(* IEC 61131-3 sources: plc_simulator/services/codesys/POUs (part 8) *)

(* ---- FB_STC_MainScheduler.st ---- *)
(* ===========================================================================================
 *  FB_STC_MainScheduler — Master scheduler orchestrator
 *
 *  Company : Galvatek part of the John Cockerill Group
 *  Author  : Jarmo Piipponen
 *  Created : 25.03.2026
 *
 * -------------------------------------------------------------------------------------------
 *  Manages FB_TSK_Scheduler and FB_DEP_Scheduler calls on
 *  alternating PLC scan cycles. Ensures they never execute
 *  on the same cycle.
 *
 *  Synchronization rules:
 *  1. Normal: alternate TSK_TURN → DEP_TURN → TSK_TURN
 *  2. Skip DEP when TSK is still computing (vPhase < 10000)
 *  3. Skip DEP when gDepPending.Valid = TRUE
 *  4. gTskStable is computed after each TSK call
 *
 *  Turn values: 0=INIT, 1=TSK_TURN, 2=DEP_TURN
 *
 *  ------------------------------------------------------------------------------------------
 *
 *  Changes:
 *
 *
 *
 *)

FUNCTION_BLOCK FB_STC_MainScheduler

(* Introduction of Variables ----------------------------------------------------------------*)

VAR_INPUT
  iRun   : BOOL;     (* TRUE = run *)
  iTimeS : LINT;     (* current absolute time (s), unix seconds *)
END_VAR

VAR_EXTERNAL CONSTANT
  MAX_UNITS     : INT;
  NOT_PROCESSED : INT;
END_VAR

VAR_EXTERNAL
  gTskStable              : BOOL;
  gConflictResolved       : BOOL;
  gDepPending             : UDT_JC_DepPendingWriteType;
  gBatch                  : ARRAY[1..MAX_UNITS] OF UDT_BatchType;
  gSchedule               : ARRAY[1..MAX_UNITS] OF UDT_JC_TskScheduleType;
  gDepWkSchedule          : ARRAY[1..MAX_UNITS] OF UDT_JC_TskScheduleType;
  (* Scheduler debug globals — written here, read by Gateway via OPC UA *)
  gSchedDbgTskPhase       : INT;
  gSchedDbgDepPhase       : INT;
  gSchedDbgTurn           : INT;
  gSchedDbgSkipCnt        : INT;
  gSchedDbgDepRejectCnt   : INT;
  gSchedDbgDepFitRound    : INT;
  gSchedDbgDepCurWaitUnit : INT;
  gSchedDbgDepWaitCnt     : INT;
  gSchedDbgBatchCnt       : INT;
  gSchedDbgTskRoundTicks  : INT;
  gSchedDbgDepRoundTicks  : INT;
END_VAR

VAR_OUTPUT
  oTskPhase : INT;     (* TSK scheduler vPhase *)
  oDepPhase : INT;     (* DEP scheduler vPhase *)
  oTurn     : INT;     (* 1=TSK ran, 2=DEP ran *)
  oSkipCnt  : INT;     (* DEP skipped count (debug) *)
END_VAR

VAR
  vFB_TskScheduler  : FB_TSK_Scheduler;
  vFB_DepScheduler  : FB_DEP_Scheduler;
  vFB_TwaCalcLimits : FB_TWA_CalcLimits;
  (* dispatch — now FC FC_STC_DispatchTask, no instance vNeeded *)
  vTurn             : INT := 0;   (* 0=init, 1=TSK, 2=DEP *)
  vSkipCnt          : INT := 0;
  vTskPhase         : INT := 0;
  vUi               : INT;
END_VAR

IF NOT iRun THEN
  (* Stop both schedulers *)
  vFB_TskScheduler(iRun := FALSE, iTimeS := 0);
  vFB_DepScheduler(iRun := FALSE, iTimeS := 0, iTskPhase := 0);
  vTurn := 0;
  vTskPhase := 0;
  oTskPhase := 0;
  oDepPhase := 0;
  oTurn := 0;
  RETURN;
END_IF;

(* ── Calculate transporter working areas (X-limits) every cycle ── *)
vFB_TwaCalcLimits();

(* ── Dispatch tasks to idle transporters (every scan) ── *)
FC_STC_DispatchTask();

(* ── Determine this cycle's vTurn ── *)
IF vTurn = 0 THEN
  (* First scan: always start with TSK *)
  vTurn := 1;

ELSIF vTurn = 1 THEN
  (* Last cycle was TSK → normally DEP's vTurn *)
  (* But skip DEP if: *)
  (*   a) TSK has not reached READY yet (vPhase < 10000) *)
  (*   b) pending data waiting for TSK to process *)
  IF vTskPhase < 10000 THEN
    (* TSK still computing — DEP would be blocked at WAIT_STABLE *)
    vTurn := 1;
    vSkipCnt := vSkipCnt + 1;
  ELSIF gDepPending.Valid THEN
    (* TSK must process pending before DEP continues *)
    vTurn := 1;
    vSkipCnt := vSkipCnt + 1;
  ELSE
    vTurn := 2;
  END_IF;

ELSIF vTurn = 2 THEN
  (* Last cycle was DEP → TSK's vTurn.
     DEP now works on sandbox arrays g_dep_wk_xxx, never live globals,
     so TSK can run freely on any cycle. *)
  vTurn := 1;
END_IF;

(* ── Execute the selected scheduler ── *)
IF vTurn = 1 THEN
  (* TSK vTurn *)
  vFB_TskScheduler(iRun := TRUE, iTimeS := iTimeS);
  vTskPhase := vFB_TskScheduler.oPhase;

  (* JS parity: set stable only when TSK reached READY and conflictResolved; do not clear here *)
    IF (vTskPhase >= 10000) AND gConflictResolved THEN
      gTskStable := TRUE;
  END_IF;

ELSIF vTurn = 2 THEN
  (* DEP vTurn *)
  vFB_DepScheduler(
    iRun       := TRUE,
    iTimeS    := iTimeS,
    iTskPhase := vTskPhase
  );
END_IF;

(* ── Publish waiting batch schedules from DEP workspace for UI display ── *)
FOR vUi := 1 TO MAX_UNITS DO
  IF gBatch[vUi].State = NOT_PROCESSED AND gDepWkSchedule[vUi].StageCount > 0 THEN
    gSchedule[vUi] := gDepWkSchedule[vUi];
  END_IF;
END_FOR;

(* ── Update outputs ── *)
oTskPhase := vFB_TskScheduler.oPhase;
oDepPhase := vFB_DepScheduler.oPhase;
oTurn      := vTurn;
oSkipCnt  := vSkipCnt;

(* ── Forward to scheduler debug globals (OPC UA readable) ── *)
gSchedDbgTskPhase        := vFB_TskScheduler.oPhase;
gSchedDbgDepPhase        := vFB_DepScheduler.oPhase;
gSchedDbgTurn             := vTurn;
gSchedDbgSkipCnt         := vSkipCnt;
gSchedDbgDepRejectCnt   := vFB_DepScheduler.oRejectCnt;
gSchedDbgDepFitRound    := vFB_DepScheduler.oFitRound;
gSchedDbgDepCurWaitUnit := vFB_DepScheduler.oCurWaitUnit;
gSchedDbgDepWaitCnt     := vFB_DepScheduler.oWaitCnt;
gSchedDbgBatchCnt        := vFB_TskScheduler.oBatchCnt;
gSchedDbgTskRoundTicks  := vFB_TskScheduler.oRoundTicks;
gSchedDbgDepRoundTicks  := vFB_DepScheduler.oRoundTicks;

END_FUNCTION_BLOCK

(* ---- FB_TSK_Scheduler.st ---- *)
(* ===========================================================================================
 *  FB_TSK_Scheduler — Main task scheduler state machine
 *
 *  Company : Galvatek part of the John Cockerill Group
 *  Author  : Jarmo Piipponen
 *  Created : 25.03.2026
 *
 * -------------------------------------------------------------------------------------------
 *  One vPhase per PLC scan cycle.
 *
 *  Phase flow (structured by 100/1000 groups):
 *  0        STOPPED
 *  1        INIT             (collect active batches)
 *  2        NO_TREATMENT_STATES
 *  1000+i   CALC_SCHEDULE    (schedule for batch i, 0..vBatchCount-1)
 *  2000     CLEAR_TASKS      (clear task queues)
 *  2001+i   CREATE_TASKS     (tasks for batch i, 0..vBatchCount-1)
 *  2100     SORT_TASKS
 *  2101     SWAP_TASKS
 *  2102     ANALYZE          (→ 2103 if vConflict, → 2200 if clean)
 *  2103     RESOLVE          (→ 2100 loop, or → 2200 if max iter)
 *  2200     NO_TREATMENT     (create no-treatment tasks)
 *  2201     APPLY_STRETCHES  (persist resolve decisions)
 *  10000    READY            (cycle complete)
 *  10001    CHECK_DEP_PENDING
 *  10002    RESTART          (→ 1)
 *
 *  Phase advancement:
 *  Default = vPhase + 1 (at end of function body).
 *  vNextPhase is set ONLY when jumping to a different group.
 *
 *  Conflict resolution: one vConflict per cycle.
 *  If resolved → back to SORT (2100).
 *  If no vConflict → NO_TREATMENT → READY.
 *  Max iterations to prevent infinite loops.
 *
 *  ------------------------------------------------------------------------------------------
 *
 *  Changes:
 *  25.03.2026 - Restructured: vPhase+1 default, vIdx from vPhase offset.
 *
 *
 *)

FUNCTION_BLOCK FB_TSK_Scheduler

(* Introduction of Variables ----------------------------------------------------------------*)

VAR_INPUT
  iRun                     : BOOL;    (* TRUE = run, FALSE = stop *)
  iTimeS                  : LINT;    (* current absolute time (s), unix seconds *)
END_VAR

VAR_EXTERNAL CONSTANT
    MAX_TRANSPORTERS        : INT;
    MAX_UNITS               : INT;
    MAX_LOCKS               : INT;
END_VAR

VAR_EXTERNAL
  g_batch                   : ARRAY[1..MAX_UNITS] OF UDT_BatchType;
  g_unit                    : ARRAY[1..MAX_UNITS] OF UDT_JC_UnitType;
  TreatmentPrograms                 : ARRAY[1..MAX_UNITS] OF UDT_TreatmentProgramType;
  g_task                    : ARRAY[1..MAX_TRANSPORTERS] OF UDT_JC_TskQueueType;
  g_schedule                : ARRAY[1..MAX_UNITS] OF UDT_JC_TskScheduleType;
  Transporters                     : ARRAY[0..MAX_TRANSPORTERS] OF UDT_TransporterType;
  (* DEP handshake *)
  g_dep_pending             : UDT_JC_DepPendingWriteType;
  g_conflict_resolved       : BOOL;
  g_tsk_stable              : BOOL;
  (* Debug observability *)
  g_dbg_tsk_conflict_type   : INT;
  g_dbg_tsk_conflict_iter   : INT;
  g_dbg_tsk_conf_unit       : INT;
  g_dbg_tsk_conf_stage      : INT;
  g_dbg_tsk_blocked_unit    : INT;
  g_dbg_tsk_blocked_stage   : INT;
  g_dbg_tsk_deficit         : DINT;
  g_dbg_tsk_stretch_cnt     : INT;
  g_dbg_tsk_total_adv       : DINT;
  g_dbg_tsk_total_delay     : DINT;
  g_dbg_prog_cal            : ARRAY[1..MAX_UNITS] OF DINT;
END_VAR

VAR_OUTPUT
  oPhase                   : INT;
  oBatchCnt               : INT;
  oTaskCnt                : INT;
  oCycleCnt               : INT;
  oConflict                : BOOL;
  oRoundTicks             : INT;     (* ticks consumed by last completed vRound *)
END_VAR

VAR
  vPhase                     : INT := 0;
  vNextPhase                : INT;
  vIdx                       : INT;    (* derived from vPhase offset *)
  (* Batch list *)
  vBatchList                : ARRAY[1..MAX_UNITS] OF INT;
  vBatchCount               : INT;
  (* Conflict iteration *)
  vConflictIter             : INT;
  MAX_CONFLICT_ITER         : INT := 40;
  (* Analyze result cache *)
  an_conflict               : BOOL;
  an_conf_type              : INT;
  an_conf_unit              : INT;
  an_conf_stage             : INT;
  an_conf_trans             : INT;
  an_blocked_unit           : INT;
  an_blocked_stage          : INT;
  an_deficit                : REAL;
  (* Resolve result cache *)
  rs_total_adv              : REAL;
  rs_total_delay            : REAL;
  (* Transporter assignment *)
  vSchedTrans               : INT;
  (* Locked stages — prevents oscillation in resolve loop *)
  vLocks                     : ARRAY[1..MAX_LOCKS] OF UDT_JC_TskLockType;
  vLockCnt                  : INT := 0;
  vLocksInitialized         : BOOL := FALSE;
  vFB_FindTransporter                   : FB_STC_FindTransporter;
  (* candidateStretches — JS: resolve decisions persisted to TreatmentPrograms *)
  vStretches                 : ARRAY[1..20] OF UDT_JC_TskStretchType;
  vStretchCnt               : INT := 0;
  si                        : INT;
  vNewCal                   : DINT;
  vFlexCap                  : DINT;
  (* Temp *)
  ui                        : INT;
  ui2                       : INT;
  ti                        : INT;
  bi                        : INT;
  vTotalTasks               : INT;
  cycle_count               : INT := 0;
  round_ticks               : INT := 0;  (* ticks since last RESTART *)
END_VAR

IF NOT iRun THEN
  IF vPhase <> 0 THEN
    FOR ti := 1 TO MAX_TRANSPORTERS DO
      g_task[ti].Count := 0;
    END_FOR;
  END_IF;
  vPhase := 0;
  oPhase := 0;
  RETURN;
END_IF;

vNextPhase := 0;
round_ticks := round_ticks + 1;

(* ══════════════════════════════════════════════════════════════ *)
(* PHASE 0: STOPPED                                             *)
(* ══════════════════════════════════════════════════════════════ *)
IF vPhase = 0 THEN
  vNextPhase := 1;

(* ══════════════════════════════════════════════════════════════ *)
(* PHASE 1: INIT — collect active batches                       *)
(* ══════════════════════════════════════════════════════════════ *)
ELSIF vPhase = 1 THEN
  (* Clear schedule for ALL units — start from clean slate *)
  FOR ui := 1 TO MAX_UNITS DO
    g_schedule[ui].StageCount := 0;
  END_FOR;
  vBatchCount := FC_STC_CollectActiveBatches(iMode := 0, oList => vBatchList);
  oBatchCnt := vBatchCount;
  vConflictIter := 0;
  vLocksInitialized := FALSE;
  vStretchCnt := 0;
  g_dbg_tsk_total_adv   := 0;
  g_dbg_tsk_total_delay := 0;

  IF vBatchCount = 0 THEN
    FOR ti := 1 TO MAX_TRANSPORTERS DO
      g_task[ti].Count := 0;
    END_FOR;
    g_conflict_resolved := TRUE;
    vNextPhase := 2200;   (* skip to NO_TREATMENT *)
  ELSE
    g_conflict_resolved := FALSE;
    (* vPhase + 1 → 2 *)
  END_IF;

(* ══════════════════════════════════════════════════════════════ *)
(* PHASE 2: NO_TREATMENT_STATES                                *)
(* ══════════════════════════════════════════════════════════════ *)
ELSIF vPhase = 2 THEN
  FC_STC_NoTreatmentStates();
  vNextPhase := 1000;

(* ══════════════════════════════════════════════════════════════ *)
(* PHASE 1000+i: CALC_SCHEDULE — one batch per scan             *)
(*   i = 0..vBatchCount-1: calculate schedule                   *)
(*   i >= vBatchCount: vDone → 2000                              *)
(* ══════════════════════════════════════════════════════════════ *)
ELSIF vPhase >= 1000 AND vPhase <= 1999 THEN
  vIdx := vPhase - 1000;

  IF vIdx < vBatchCount THEN
    ui := vBatchList[vIdx + 1];

    (* CalcSchedule handles elapsed-time normalisation — no pre-adjustment vNeeded here. *)

    IF g_unit[ui].vLocation < MIN_STATION_INDEX THEN
      vSchedTrans := g_unit[ui].vLocation;
    ELSE
      vFB_FindTransporter(iLiftStn := g_unit[ui].vLocation, iSinkStn := 0);
      vSchedTrans := vFB_FindTransporter.oTrans;
      IF vSchedTrans = 0 THEN vSchedTrans := 1; END_IF;
    END_IF;

    FC_STC_CalcSchedule(iUnit := ui, iTrans := vSchedTrans, iTimeS := iTimeS,
                     ioSchedule := g_schedule, ioBatch := g_batch, ioProgram := TreatmentPrograms);
    (* vPhase + 1 → next batch *)

  ELSE
    vNextPhase := 2000;
  END_IF;

(* ══════════════════════════════════════════════════════════════ *)
(* PHASE 2000: CLEAR_TASKS — clear all task queues              *)
(* ══════════════════════════════════════════════════════════════ *)
ELSIF vPhase = 2000 THEN
  FOR ti := 1 TO MAX_TRANSPORTERS DO
    g_task[ti].Count := 0;
  END_FOR;
  (* vPhase + 1 → 2001 *)

(* ══════════════════════════════════════════════════════════════ *)
(* PHASE 2001+i: CREATE_TASKS — one batch per scan              *)
(*   i = 0..vBatchCount-1: create tasks                         *)
(*   i >= vBatchCount: vDone → 2100                              *)
(* ══════════════════════════════════════════════════════════════ *)
ELSIF vPhase >= 2001 AND vPhase <= 2099 THEN
  vIdx := vPhase - 2001;

  IF vIdx < vBatchCount THEN
    ui := vBatchList[vIdx + 1];
    FC_STC_CreateTasks(iUnit := ui, ioSchedule := g_schedule, ioTask := g_task);
    (* vPhase + 1 → next batch *)
  ELSE
    vNextPhase := 2100;
  END_IF;

(* ══════════════════════════════════════════════════════════════ *)
(* PHASE 2100: SORT_TASKS                                       *)
(* ══════════════════════════════════════════════════════════════ *)
ELSIF vPhase = 2100 THEN
  FC_STC_SortTasks(iTrans := 0, iTimeS := iTimeS, ioTask := g_task, ioBatch := g_batch);
  IF NOT vLocksInitialized THEN
    vLockCnt := 0;
    FOR bi := 1 TO MAX_LOCKS DO
      vLocks[bi].Unit := 0;
      vLocks[bi].Stage := 0;
      vLocks[bi].Direction := 0;
    END_FOR;
    vLocksInitialized := TRUE;
  END_IF;
  (* vPhase + 1 → 2101 *)

(* ══════════════════════════════════════════════════════════════ *)
(* PHASE 2101: SWAP_TASKS                                       *)
(* ══════════════════════════════════════════════════════════════ *)
ELSIF vPhase = 2101 THEN
  FC_STC_SwapTasks(ioTask := g_task);
  (* vPhase + 1 → 2102 *)

(* ══════════════════════════════════════════════════════════════ *)
(* PHASE 2102: ANALYZE                                          *)
(* ══════════════════════════════════════════════════════════════ *)
ELSIF vPhase = 2102 THEN
  FC_TSK_Analyze(ioTask := g_task,
    oHasConflict => an_conflict, oConfType => an_conf_type,
    oConfUnit => an_conf_unit, oConfStage => an_conf_stage,
    oConfTrans => an_conf_trans, oBlockedUnit => an_blocked_unit,
    oBlockedStage => an_blocked_stage, oDeficit => an_deficit);
  oConflict := an_conflict;

  IF an_conflict THEN
    g_dbg_tsk_conflict_type  := an_conf_type;
    g_dbg_tsk_conf_unit      := an_conf_unit;
    g_dbg_tsk_conf_stage     := an_conf_stage;
    g_dbg_tsk_blocked_unit   := an_blocked_unit;
    g_dbg_tsk_blocked_stage  := an_blocked_stage;
    g_dbg_tsk_deficit        := REAL_TO_DINT(an_deficit);
    g_conflict_resolved := FALSE;
    (* vPhase + 1 → 2103 RESOLVE *)
  ELSE
    g_conflict_resolved := TRUE;
    vNextPhase := 2200;   (* skip RESOLVE → NO_TREATMENT *)
  END_IF;

(* ══════════════════════════════════════════════════════════════ *)
(* PHASE 2103: RESOLVE — one vConflict, then re-analyze          *)
(* ══════════════════════════════════════════════════════════════ *)
ELSIF vPhase = 2103 THEN
  FC_TSK_Resolve(
    iConfUnit     := an_conf_unit,
    iConfStage    := an_conf_stage,
    iConfTrans    := an_conf_trans,
    iBlockedUnit  := an_blocked_unit,
    iBlockedStage := an_blocked_stage,
    iDeficit       := an_deficit,
    ioLocks        := vLocks,
    ioLockCnt     := vLockCnt,
    ioSchedule     := g_schedule,
    ioTask         := g_task,
    ioBatch        := g_batch,
    oTotalAdv     => rs_total_adv,
    oTotalDelay   => rs_total_delay
  );

  (* Collect vStretches *)
  IF rs_total_adv > 0.1 AND vStretchCnt < 20 THEN
    vStretchCnt := vStretchCnt + 1;
    vStretches[vStretchCnt].Unit   := an_blocked_unit;
    vStretches[vStretchCnt].Stage  := an_blocked_stage;
    vStretches[vStretchCnt].DelayS := -REAL_TO_DINT(rs_total_adv);
    g_dbg_tsk_total_adv := g_dbg_tsk_total_adv + REAL_TO_DINT(rs_total_adv);
  END_IF;
  IF rs_total_delay > 0.1 AND vStretchCnt < 20 THEN
    vStretchCnt := vStretchCnt + 1;
    vStretches[vStretchCnt].Unit   := an_conf_unit;
    vStretches[vStretchCnt].Stage  := an_conf_stage;
    vStretches[vStretchCnt].DelayS := REAL_TO_DINT(rs_total_delay);
    g_dbg_tsk_total_delay := g_dbg_tsk_total_delay + REAL_TO_DINT(rs_total_delay);
  END_IF;

  vConflictIter := vConflictIter + 1;

  IF vConflictIter >= MAX_CONFLICT_ITER THEN
    g_conflict_resolved := TRUE;
    vNextPhase := 2200;   (* accept partial, move on *)
  ELSE
    vNextPhase := 2100;   (* re-SORT → SWAP → ANALYZE *)
  END_IF;

(* ══════════════════════════════════════════════════════════════ *)
(* PHASE 2200: NO_TREATMENT — create no-treatment tasks         *)
(* ══════════════════════════════════════════════════════════════ *)
ELSIF vPhase = 2200 THEN
  FC_STC_ManualTask(iTimeS := iTimeS, ioTask := g_task);
  FC_TSK_NoTreatment(iTimeS := iTimeS, ioTask := g_task);
  oConflict := FALSE;
  (* vPhase + 1 → 2201 *)

(* ══════════════════════════════════════════════════════════════ *)
(* PHASE 2201: APPLY_STRETCHES — persist resolve decisions      *)
(* ══════════════════════════════════════════════════════════════ *)
ELSIF vPhase = 2201 THEN
  FOR si := 1 TO vStretchCnt DO
    IF vStretches[si].Unit >= 1 AND vStretches[si].Unit <= MAX_UNITS THEN
     IF vStretches[si].Stage >= 1
        AND vStretches[si].Stage <= TreatmentPrograms[vStretches[si].Unit].StepCount THEN
      vNewCal := TreatmentPrograms[vStretches[si].Unit].Steps[vStretches[si].Stage].CalTime
               + vStretches[si].DelayS;
      IF vNewCal < TreatmentPrograms[vStretches[si].Unit].Steps[vStretches[si].Stage].MinTime THEN
        vNewCal := TreatmentPrograms[vStretches[si].Unit].Steps[vStretches[si].Stage].MinTime;
      END_IF;
      (* Flex cap: min + factor × (max - min) *)
      vFlexCap := TreatmentPrograms[vStretches[si].Unit].Steps[vStretches[si].Stage].MinTime
               + REAL_TO_DINT(SCH_TSK_FLEX_FACTOR * DINT_TO_REAL(
                   TreatmentPrograms[vStretches[si].Unit].Steps[vStretches[si].Stage].MaxTime
                 - TreatmentPrograms[vStretches[si].Unit].Steps[vStretches[si].Stage].MinTime));
      IF vNewCal > vFlexCap THEN
        vNewCal := vFlexCap;
      END_IF;
      TreatmentPrograms[vStretches[si].Unit].Steps[vStretches[si].Stage].CalTime := vNewCal;

      IF g_batch[vStretches[si].Unit].CurStage = vStretches[si].Stage THEN
        g_batch[vStretches[si].Unit].CalTime := vNewCal;
      END_IF;
     END_IF;
    END_IF;
  END_FOR;
  vStretchCnt := 0;
  (* vPhase + 1 → 2202 *)

(* ══════════════════════════════════════════════════════════════ *)
(* PHASE 2202: MOVE_AWAY — idle transporter move-away check     *)
(* ══════════════════════════════════════════════════════════════ *)
ELSIF vPhase = 2202 THEN
  FC_STC_TakeOut(iTimeS := iTimeS);
  vNextPhase := 10000;

(* ══════════════════════════════════════════════════════════════ *)
(* PHASE 10000: READY — cycle complete                          *)
(* ══════════════════════════════════════════════════════════════ *)
ELSIF vPhase = 10000 THEN
  vTotalTasks := 0;
  FOR ti := 1 TO MAX_TRANSPORTERS DO
    vTotalTasks := vTotalTasks + g_task[ti].Count;
  END_FOR;
  oTaskCnt := vTotalTasks;

  IF NOT oConflict THEN
    g_dbg_tsk_conflict_type := 0;
    g_dbg_tsk_conf_unit     := 0;
    g_dbg_tsk_conf_stage    := 0;
    g_dbg_tsk_blocked_unit  := 0;
    g_dbg_tsk_blocked_stage := 0;
    g_dbg_tsk_deficit       := 0;
  END_IF;
  g_dbg_tsk_conflict_iter := vConflictIter;
  g_dbg_tsk_stretch_cnt   := vStretchCnt;

  FOR ui := 1 TO MAX_UNITS DO
    IF g_batch[ui].CurStage >= 1
       AND g_batch[ui].CurStage <= TreatmentPrograms[ui].StepCount THEN
      g_dbg_prog_cal[ui] := TreatmentPrograms[ui].Steps[g_batch[ui].CurStage].CalTime;
    ELSE
      g_dbg_prog_cal[ui] := 0;
    END_IF;
  END_FOR;
  (* vPhase + 1 → 10001 *)

(* ══════════════════════════════════════════════════════════════ *)
(* PHASE 10001: CHECK_DEP_PENDING                               *)
(* ══════════════════════════════════════════════════════════════ *)
ELSIF vPhase = 10001 THEN
  IF g_dep_pending.Valid THEN
    FOR ui := 1 TO MAX_UNITS DO
      IF g_dep_pending.Programs[ui].ProgramId > 0 THEN
        TreatmentPrograms[ui] := g_dep_pending.Programs[ui];
      END_IF;
    END_FOR;
    IF g_dep_pending.BatchUnit >= 1 AND g_dep_pending.BatchUnit <= MAX_UNITS THEN
      g_batch[g_dep_pending.BatchUnit].CurStage   := g_dep_pending.BatchStage;
      g_batch[g_dep_pending.BatchUnit].State       := g_dep_pending.BatchState;
      g_batch[g_dep_pending.BatchUnit].StartTime   := g_dep_pending.TimeStamp;
      g_batch[g_dep_pending.BatchUnit].MinTime     := g_dep_pending.BatchMinTime;
      g_batch[g_dep_pending.BatchUnit].MaxTime     := g_dep_pending.BatchMaxTime;
      g_batch[g_dep_pending.BatchUnit].CalTime     := g_dep_pending.BatchCalTime;
    END_IF;
    (* Apply active batch CalTimes written by DEP *)
    FOR ui := 1 TO MAX_UNITS DO
      IF g_dep_pending.ActiveBatchCalTime[ui] > 0
         AND ui <> g_dep_pending.BatchUnit THEN
        g_batch[ui].CalTime := g_dep_pending.ActiveBatchCalTime[ui];
      END_IF;
    END_FOR;
    g_dep_pending.Valid := FALSE;
    g_conflict_resolved := FALSE;
    g_tsk_stable := FALSE;
    vNextPhase := 1;   (* full recalculation *)
  END_IF;
  (* else vPhase + 1 → 10002 *)

(* ══════════════════════════════════════════════════════════════ *)
(* PHASE 10002: RESTART — begin new cycle                       *)
(* ══════════════════════════════════════════════════════════════ *)
ELSIF vPhase = 10002 THEN
  cycle_count := cycle_count + 1;
  oCycleCnt := cycle_count;
  oRoundTicks := round_ticks;
  round_ticks := 0;
  vNextPhase := 1;

(* ══════════════════════════════════════════════════════════════ *)
(* Unknown vPhase → reset                                        *)
(* ══════════════════════════════════════════════════════════════ *)
ELSE
  vNextPhase := 1;
END_IF;

(* ── Phase advancement: default = vPhase + 1 ── *)
IF vNextPhase > 0 THEN
  vPhase := vNextPhase;
ELSE
  vPhase := vPhase + 1;
END_IF;
oPhase := vPhase;

END_FUNCTION_BLOCK

(* ---- FB_TWA_CalcLimits.st ---- *)
(* ===========================================================================================
 *  FB_TWA_CalcLimits — Transporter Working Area: X-limit calculation
 *
 *  Company : Galvatek part of the John Cockerill Group
 *  Author  : Jarmo Piipponen
 *  Created : 25.03.2026
 *
 * -------------------------------------------------------------------------------------------
 *  Calculates x_min_limit and x_max_limit for all active
 *  transporters. Collision avoidance layers:
 *
 *  Pass 1 (per transporter):
 *  - Station restrictions from gAvoidStatus
 *  - Safety vDistance from same-line neighbors
 *  - canEvade, vPriority, x-vRank computation
 *
 *  Pass 2 (pair comparisons):
 *  - Priority-based restrictions (higher → lower)
 *  - Bidirectional safety (same direction chase)
 *
 *  Final: Trap validation
 *
 *  ------------------------------------------------------------------------------------------
 *
 *  Changes:
 *
 *
 *
 *)

FUNCTION_BLOCK FB_TWA_CalcLimits

(* Introduction of Variables ----------------------------------------------------------------*)

VAR_EXTERNAL CONSTANT
    MAX_TRANSPORTERS  : INT;
    MAX_UNITS         : INT;
    MIN_STATION_INDEX : INT;
    MAX_STATION_INDEX : INT;
    AVOID_PASSABLE    : INT;
    AVOID_BLOCK       : INT;
    MIN_WORKING_AREA  : DINT;
    IN_PROCESS        : INT;
END_VAR

VAR_EXTERNAL
  Transporters      : ARRAY[0..MAX_TRANSPORTERS] OF UDT_TransporterType;
  gTransporter      : ARRAY[1..MAX_TRANSPORTERS] OF UDT_TransporterStatusType;
  Stations          : ARRAY[MIN_STATION_INDEX..MAX_STATION_INDEX] OF UDT_StationType;
  CountStations     : INT;
  gAvoidStatus      : ARRAY[MIN_STATION_INDEX..MAX_STATION_INDEX] OF INT;
  gStationOccupancy : ARRAY[1..MAX_STATION_INDEX] OF UDT_JC_UnitAtStationType;
  gBatch            : ARRAY[1..MAX_UNITS] OF UDT_BatchType;
END_VAR

VAR
  i             : INT;
  j             : INT;
  vStnNum       : INT;
  vStnX         : DINT;
  vAvoidSt      : INT;
  vMinX         : DINT;
  vMaxX         : DINT;
  vCurrentX     : DINT;
  vCurrentY     : DINT;
  vAvoidDist    : DINT;
  vIsTarget     : BOOL;
  vNewVal       : DINT;

  (* Station scan: nearest restricting station per side *)
  vNearLeftX    : DINT;
  vNearLeftStn  : INT;
  vNearRightX   : DINT;
  vNearRightStn : INT;
  vHasLeft      : BOOL;
  vHasRight     : BOOL;
  vMidpoint     : DINT;

  (* Per-transporter computed values *)
  vPriority     : ARRAY[1..MAX_TRANSPORTERS] OF DINT;
  vCanEvade     : ARRAY[1..MAX_TRANSPORTERS] OF BOOL;
  vRank         : ARRAY[1..MAX_TRANSPORTERS] OF INT;

  (* Pair comparison *)
  vOtherX       : DINT;
  vOtherY       : DINT;
  vIPhase       : INT;
  vJPhase       : INT;
  vDist         : DINT;
  vWorkArea     : DINT;
  vAWins        : BOOL;
  vRestrictX    : DINT;
  vBetween      : INT;
  vChainOfs     : DINT;
  vAdjusted     : DINT;

  (* Bidirectional *)
  vIMovingRight : BOOL;
  vIMovingLeft  : BOOL;
  vJMovingRight : BOOL;
  vJMovingLeft  : BOOL;

  (* IN_PROCESS batch vPriority boost *)
  vLiftStn      : INT;
  vLiftUid      : INT;
  vBatchBoost   : DINT;

  (* Full task extent for vRestrictX *)
  vLiftX        : DINT;
  vSinkX        : DINT;
  vILiftStn     : INT;
  vISinkStn     : INT;
END_VAR

(* ══════════════════════════════════════════════════════════════
   PASS 1: Station restrictions + safety vDistance + properties
   Each transporter computes its OWN limits in one iteration.
   ══════════════════════════════════════════════════════════════ *)
FOR i := 1 TO MAX_TRANSPORTERS DO
  IF NOT gTransporter[i].IsActive THEN
    vPriority[i] := 0;
    vCanEvade[i] := FALSE;
    vRank[i] := 0;
    CONTINUE;
  END_IF;

  vMinX := Transporters[i].DrivePosMin;
  vMaxX := Transporters[i].DrivePosMax;
  vCurrentX := gTransporter[i].XPosition;
  vCurrentY := gTransporter[i].YPosition;
  vAvoidDist := Transporters[i].AvoidanceWidth;

  (* Lock transporters with no drive range configured *)
  IF (vMinX < 1) OR (vMaxX < 1) THEN
    gTransporter[i].XMinDriveLimit := vCurrentX;
    gTransporter[i].XMaxDriveLimit := vCurrentX;
    vPriority[i] := 0;
    vCanEvade[i] := FALSE;
    vRank[i] := 0;
    CONTINUE;
  END_IF;

  (* ── Station scan: find nearest restrict LEFT and RIGHT ──────
     Single pass through all stations. Only Block and
     Passable-target stations cause restrictions. *)
  vHasLeft := FALSE;
  vHasRight := FALSE;
  vNearLeftX := 0;
  vNearLeftStn := 0;
  vNearRightX := 0;
  vNearRightStn := 0;

  FOR vStnNum := MIN_STATION_INDEX TO MAX_STATION_INDEX DO
    IF Stations[vStnNum].TankId = 0 THEN CONTINUE; END_IF;

    vAvoidSt := gAvoidStatus[vStnNum];
    IF vAvoidSt = 0 THEN CONTINUE; END_IF;  (* AVOID_NONE *)

    (* Passable: only restricts if this transporter's target *)
    IF vAvoidSt = AVOID_PASSABLE THEN
      vIsTarget := (vStnNum = gTransporter[i].LiftStationTarget)
               OR  (vStnNum = gTransporter[i].SinkStationTarget);
      IF NOT vIsTarget THEN CONTINUE; END_IF;
    END_IF;

    (* Station is Block or Passable+target → track nearest per side *)
    vStnX := Stations[vStnNum].XPosition;

    IF vStnX < vCurrentX THEN
      IF NOT vHasLeft OR vStnX > vNearLeftX THEN
        vNearLeftX := vStnX;
        vNearLeftStn := vStnNum;
        vHasLeft := TRUE;
      END_IF;
    ELSIF vStnX > vCurrentX THEN
      IF NOT vHasRight OR vStnX < vNearRightX THEN
        vNearRightX := vStnX;
        vNearRightStn := vStnNum;
        vHasRight := TRUE;
      END_IF;
    END_IF;
  END_FOR;

  (* Apply station restrictions using station-specific AvoidDistance *)
  IF vHasLeft THEN
    vNewVal := vNearLeftX + Stations[vNearLeftStn].AvoidDistance;
    IF vNewVal > vMinX THEN vMinX := vNewVal; END_IF;
  END_IF;
  IF vHasRight THEN
    vNewVal := vNearRightX - Stations[vNearRightStn].AvoidDistance;
    IF vNewVal < vMaxX THEN vMaxX := vNewVal; END_IF;
  END_IF;

  (* Conflict: trapped vBetween two restricting stations *)
  IF (vMinX >= vMaxX) AND vHasLeft AND vHasRight THEN
    vMidpoint := (vNearLeftX + vNearRightX) / 2;
    vMinX := vMidpoint - 5;
    vMaxX := vMidpoint + 5;
  END_IF;

  (* ── Safety vDistance: each same-line neighbor pushes i away ── *)
  FOR j := 1 TO MAX_TRANSPORTERS DO
    IF j = i THEN CONTINUE; END_IF;
    IF NOT gTransporter[j].IsActive THEN CONTINUE; END_IF;

    vOtherY := gTransporter[j].YPosition;
    IF ABS(vOtherY - vCurrentY) >= 1 THEN CONTINUE; END_IF;

    vOtherX := gTransporter[j].XPosition;

    IF vOtherX < vCurrentX THEN
      (* j is LEFT → j's safety zone pushes i's min up *)
      vNewVal := vOtherX + Transporters[j].AvoidanceWidth;
  IF vNewVal > vMinX THEN vMinX := vNewVal; END_IF;
    ELSIF vOtherX > vCurrentX THEN
      (* j is RIGHT → j's safety zone pushes i's max down *)
      vNewVal := vOtherX - Transporters[j].AvoidanceWidth;
  IF vNewVal < vMaxX THEN vMaxX := vNewVal; END_IF;
    END_IF;
  END_FOR;

  (* ── Write limits ── *)
  gTransporter[i].XMinDriveLimit := vMinX;
  gTransporter[i].XMaxDriveLimit := vMaxX;

  (* ── canEvade (inline) ── *)
  vCanEvade[i] := TRUE;
  IF gTransporter[i].Status < 3 THEN
    vCanEvade[i] := FALSE;
  END_IF;
  IF (gTransporter[i].Status = 4)
     AND ((gTransporter[i].Phase = 2) OR (gTransporter[i].Phase = 4)) THEN
    vCanEvade[i] := FALSE;
  END_IF;
  vWorkArea := vMaxX - vMinX;
  IF vWorkArea < MIN_WORKING_AREA THEN
    vCanEvade[i] := FALSE;
  END_IF;

  (* ── Priority (inline, replaces TWA_CalcPriority call) ──────
     IN_PROCESS batch boost: +100000 if the task serves an
     IN_PROCESS batch. Phases 1-4 all check via LiftStation
     unit lookup (unit stays associated throughout transfer).
     This ensures treatment tasks trump NTT/empty moves. ── *)
  vIPhase := gTransporter[i].Phase;
  vBatchBoost := 0;
  IF vIPhase >= 1 AND vIPhase <= 4 THEN
    vLiftStn := gTransporter[i].LiftStationTarget;
    IF vLiftStn >= 1 AND vLiftStn <= MAX_STATION_INDEX THEN
      vLiftUid := gStationOccupancy[vLiftStn].UnitId;
      IF vLiftUid >= 1 AND vLiftUid <= MAX_UNITS THEN
        IF gBatch[vLiftUid].State = IN_PROCESS THEN
          vBatchBoost := DINT#100000;
        END_IF;
      END_IF;
    END_IF;
  END_IF;

  IF NOT vCanEvade[i] THEN
    vPriority[i] := DINT#100000;
  ELSIF vIPhase = 3 OR vIPhase = 4 THEN
    vDist := ABS(vCurrentX - gTransporter[i].XFinalTarget);
  IF vDist > 99999 THEN vDist := 99999; END_IF;
    vPriority[i] := DINT#200000 + vBatchBoost + (DINT#99999 - vDist);
  ELSIF vIPhase = 1 OR vIPhase = 2 THEN
    (* Move-away (Status=3, Phase=1) gets idle-class vPriority, not active-task vPriority *)
    IF gTransporter[i].Status = 3 THEN
      vPriority[i] := 2;  (* above stationary idle (1), below active tasks (100000+) *)
    ELSE
      vDist := ABS(vCurrentX - gTransporter[i].XFinalTarget);
      IF vDist > 99999 THEN vDist := 99999; END_IF;
      vPriority[i] := DINT#100000 + vBatchBoost + (DINT#99999 - vDist);
    END_IF;
  ELSE
    vPriority[i] := 1;
  END_IF;

  (* ── X-vRank among same-line active transporters ──
     vRank = 1 + count of same-line transporters with smaller x *)
  vRank[i] := 1;
  FOR j := 1 TO MAX_TRANSPORTERS DO
    IF j = i THEN CONTINUE; END_IF;
    IF NOT gTransporter[j].IsActive THEN CONTINUE; END_IF;
    IF ABS(gTransporter[j].YPosition - vCurrentY) >= 1 THEN CONTINUE; END_IF;
    IF gTransporter[j].XPosition < vCurrentX THEN
      vRank[i] := vRank[i] + 1;
    END_IF;
  END_FOR;
END_FOR;

(* ══════════════════════════════════════════════════════════════
   PASS 2: Priority restrictions + bidirectional safety
   Each pair (i,j): i restricts j if i has higher vPriority.
   ══════════════════════════════════════════════════════════════ *)
FOR i := 1 TO MAX_TRANSPORTERS DO
  IF NOT gTransporter[i].IsActive THEN CONTINUE; END_IF;
  IF vPriority[i] = 0 THEN CONTINUE; END_IF;

  vCurrentX := gTransporter[i].XPosition;
  vCurrentY := gTransporter[i].YPosition;
  vIPhase := gTransporter[i].Phase;

  FOR j := 1 TO MAX_TRANSPORTERS DO
    IF j = i THEN CONTINUE; END_IF;
    IF NOT gTransporter[j].IsActive THEN CONTINUE; END_IF;
    IF vPriority[j] = 0 THEN CONTINUE; END_IF;

    vOtherY := gTransporter[j].YPosition;
    IF ABS(vOtherY - vCurrentY) >= 1 THEN CONTINUE; END_IF;

    vOtherX := gTransporter[j].XPosition;
    vJPhase := gTransporter[j].Phase;

    (* ── Priority restrictions: i restricts j if i wins ── *)
    (* Move-away (Status=3, Phase=1) participates in restrictions
       so it can push stationary idle transporters out of its way *)
    IF (vIPhase <> 0) OR (gTransporter[i].Status = 3 AND vIPhase = 1) THEN
      vAWins := FALSE;
      IF vPriority[i] > vPriority[j] THEN
        vAWins := TRUE;
      ELSIF (vPriority[i] = vPriority[j]) AND (i < j) THEN
        vAWins := TRUE;
      END_IF;

      IF vAWins THEN
        (* Full task extent: use the extreme position
           of both lift and sink stations on the side
           facing j. This prevents j from first driving
           closer and then having to reverse when i
           moves to the other end of its task. *)
        vILiftStn := gTransporter[i].LiftStationTarget;
        vISinkStn := gTransporter[i].SinkStationTarget;
        IF vIPhase >= 1 AND vIPhase <= 4 THEN
          vLiftX := vCurrentX;
          vSinkX := vCurrentX;
          IF vILiftStn >= MIN_STATION_INDEX
             AND vILiftStn <= MAX_STATION_INDEX THEN
            vLiftX := Stations[vILiftStn].XPosition;
          END_IF;
          IF vISinkStn >= MIN_STATION_INDEX
             AND vISinkStn <= MAX_STATION_INDEX THEN
            vSinkX := Stations[vISinkStn].XPosition;
          END_IF;
          IF vCurrentX < vOtherX THEN
            (* i LEFT of j → use rightmost extent *)
            vRestrictX := vLiftX;
            IF vSinkX > vRestrictX THEN
              vRestrictX := vSinkX;
            END_IF;
            IF vCurrentX > vRestrictX THEN
              vRestrictX := vCurrentX;
            END_IF;
          ELSE
            (* i RIGHT of j → use leftmost extent *)
            vRestrictX := vLiftX;
            IF vSinkX < vRestrictX THEN
              vRestrictX := vSinkX;
            END_IF;
            IF vCurrentX < vRestrictX THEN
              vRestrictX := vCurrentX;
            END_IF;
          END_IF;
        ELSE
          vRestrictX := vCurrentX;
        END_IF;

        (* "vBetween" from pre-computed vRank *)
        vBetween := ABS(vRank[i] - vRank[j]) - 1;
  IF vBetween < 0 THEN vBetween := 0; END_IF;

        vChainOfs := Transporters[i].AvoidanceWidth
                   + INT_TO_DINT(vBetween) * (MIN_WORKING_AREA + Transporters[i].AvoidanceWidth);

        IF vCurrentX < vOtherX THEN
          (* i LEFT, j RIGHT → restrict j's XMin *)
          vNewVal := vRestrictX + vChainOfs;
          IF vNewVal > gTransporter[j].XMinDriveLimit THEN
            IF vNewVal <= (gTransporter[j].XMaxDriveLimit - MIN_WORKING_AREA) THEN
              gTransporter[j].XMinDriveLimit := vNewVal;
            ELSE
              vAdjusted := gTransporter[j].XMaxDriveLimit - MIN_WORKING_AREA;
              IF vAdjusted > gTransporter[j].XMinDriveLimit THEN
                gTransporter[j].XMinDriveLimit := vAdjusted;
              END_IF;
            END_IF;
          END_IF;

        ELSIF vCurrentX > vOtherX THEN
          (* i RIGHT, j LEFT → restrict j's XMax *)
          vNewVal := vRestrictX - vChainOfs;
          IF vNewVal < gTransporter[j].XMaxDriveLimit THEN
            IF vNewVal >= (gTransporter[j].XMinDriveLimit + MIN_WORKING_AREA) THEN
              gTransporter[j].XMaxDriveLimit := vNewVal;
            ELSE
              vAdjusted := gTransporter[j].XMinDriveLimit + MIN_WORKING_AREA;
              IF vAdjusted < gTransporter[j].XMaxDriveLimit THEN
                gTransporter[j].XMaxDriveLimit := vAdjusted;
              END_IF;
            END_IF;
          END_IF;
        END_IF;
      END_IF;
    END_IF;

    (* ── Bidirectional safety: only adjacent (vRank diff = 1) ── *)
    IF ABS(vRank[i] - vRank[j]) = 1 THEN
      vIMovingRight := ((vIPhase = 1) OR (vIPhase = 3))
                        AND (gTransporter[i].XFinalTarget > vCurrentX);
      vJMovingRight := ((vJPhase = 1) OR (vJPhase = 3))
                        AND (gTransporter[j].XFinalTarget > vOtherX);
      vIMovingLeft := ((vIPhase = 1) OR (vIPhase = 3))
                       AND (gTransporter[i].XFinalTarget < vCurrentX);
      vJMovingLeft := ((vJPhase = 1) OR (vJPhase = 3))
                       AND (gTransporter[j].XFinalTarget < vOtherX);

      IF vCurrentX < vOtherX AND vIMovingRight AND vJMovingRight THEN
        (* i LEFT chasing j RIGHT → restrict j's XMin *)
        vNewVal := vCurrentX + Transporters[i].AvoidanceWidth;
        IF vNewVal > gTransporter[j].XMinDriveLimit THEN
          gTransporter[j].XMinDriveLimit := vNewVal;
        END_IF;
      END_IF;

      IF vCurrentX > vOtherX AND vIMovingLeft AND vJMovingLeft THEN
        (* i RIGHT chasing j LEFT → restrict j's XMax *)
        vNewVal := vCurrentX - Transporters[i].AvoidanceWidth;
        IF vNewVal < gTransporter[j].XMaxDriveLimit THEN
          gTransporter[j].XMaxDriveLimit := vNewVal;
        END_IF;
      END_IF;
    END_IF;
  END_FOR;
END_FOR;

(* ══════════════════════════════════════════════════════════════
   TRAP VALIDATION: if restrictions vConflict, lock in place
   ══════════════════════════════════════════════════════════════ *)
FOR i := 1 TO MAX_TRANSPORTERS DO
  IF NOT gTransporter[i].IsActive THEN CONTINUE; END_IF;
  IF gTransporter[i].XMinDriveLimit > gTransporter[i].XMaxDriveLimit THEN
    gTransporter[i].XMinDriveLimit := gTransporter[i].XPosition;
    gTransporter[i].XMaxDriveLimit := gTransporter[i].XPosition;
  END_IF;
END_FOR;

END_FUNCTION_BLOCK

(* ---- SIM_FB_ClearConfig.st ---- *)
(* ============================================================
   SIM_FB_ClearConfig.st — Clear all PLC configuration data

   Called by PLC_PRG when Gateway sends cmd=3 (clear_all).
   Zeroes out all stations, transporter configs, transporter
   states and units so the PLC is ready for fresh config upload.
   ============================================================ *)

FUNCTION_BLOCK SIM_FB_ClearConfig
VAR_EXTERNAL CONSTANT
    MAX_Transporters    : INT;
    MAX_STATIONS_PER_STEP       : INT;
    MIN_StationIndex : INT;
    MAX_StationIndex   : INT;
    MAX_Units           : INT;
    DEP_MAX_WAITING     : INT;
END_VAR

VAR_EXTERNAL
  g_station_count    : INT;
  g_station         : ARRAY[MIN_StationIndex..MAX_StationIndex] OF UDT_StationType;
  g_station_loc     : ARRAY[1..MAX_StationIndex] OF UDT_UnitLocation;
  g_cfg              : ARRAY[1..MAX_Transporters] OF UDT_TransporterType;
  g_transporter      : ARRAY[1..MAX_Transporters] OF UDT_TransporterStatusType;
  g_sim_trans        : ARRAY[1..MAX_Transporters] OF UDT_JC_SimTransporterType;
  g_unit            : ARRAY[1..MAX_Units] OF UDT_UnitType;
  g_ntt             : ARRAY[1..MAX_Transporters] OF UDT_JC_NttTransporterType;
  g_batch          : ARRAY[1..MAX_Units] OF UDT_BatchType;
  g_program         : ARRAY[1..MAX_Units] OF UDT_TreatmentProgramType;
  g_avoid_status     : ARRAY[MIN_StationIndex..MAX_StationIndex] OF INT;
  g_schedule         : ARRAY[1..MAX_Units] OF UDT_JC_TskScheduleType;
  g_task             : ARRAY[1..MAX_Transporters] OF UDT_JC_TskQueueType;
  g_dep_sandbox      : UDT_JC_DepSandboxType;
  g_dep_pending      : UDT_JC_DepPendingWriteType;
  g_dep_activated    : BOOL;
  g_tsk_stable       : BOOL;
  g_dep_waiting_count : INT;
  g_dep_waiting       : ARRAY[1..DEP_MAX_WAITING] OF INT;
  g_dep_wait_unit     : INT;
END_VAR
VAR
  i : INT;
  j : INT;
  k : INT;
END_VAR

(* --- Clear all stations --- *)
FOR i := MIN_StationIndex TO MAX_StationIndex DO
  g_station[i].TankId       := 0;
  g_station[i].IsInUse       := FALSE;
  g_station[i].XPosition    := 0;
  g_station[i].YPosition    := 0;
  g_station[i].ZPosition    := 0;
  g_station[i].DryWet          := 0;
  g_station[i].StationType     := 0;
  g_station[i].DrippingTime := 0;
  g_station[i].DeviceDelay  := 0;
END_FOR;

(* --- Clear all location tracking (transporters 1..MAX_Transporters + stations MIN..MAX) --- *)
FOR i := 1 TO MAX_StationIndex DO
  g_station_loc[i].UnitId     := 0;
  g_station_loc[i].ChangeTime := 0;
END_FOR;
g_station_count := 0;

(* --- Clear all transporter configs --- *)
FOR i := 1 TO MAX_Transporters DO
  g_cfg[i].DrivePosMin   := 0;
  g_cfg[i].DrivePosMax   := 0;
  g_cfg[i].YMinDriveLimit   := 0;
  g_cfg[i].YMaxDriveLimit   := 0;
  g_cfg[i].CollisionWidth    := 0;
  g_cfg[i].AvoidanceWidth    := 0;
  g_cfg[i].Acceleration_X     := 0;
  g_cfg[i].Deceleration_X     := 0;
  g_cfg[i].SpeedMax_X    := 0;
  g_cfg[i].ZPosDown    := 0;
  g_cfg[i].ZPosSlowUp := 0;
  g_cfg[i].ZPosSlowDown := 0;
  g_cfg[i].ZPosSlowEnd := 0;
  g_cfg[i].SpeedLiftSlow_Z   := 0;
  g_cfg[i].SpeedLiftFast_Z   := 0;
  g_cfg[i].DripTrayDelay  := 0;
  FOR j := 1 TO 4 DO
    g_cfg[i].TaskArea[j].MinLift := 0;
    g_cfg[i].TaskArea[j].MaxLift := 0;
    g_cfg[i].TaskArea[j].MinSink := 0;
    g_cfg[i].TaskArea[j].MaxSink := 0;
  END_FOR;
END_FOR;

(* --- Clear avoid status --- *)
FOR i := MIN_StationIndex TO MAX_StationIndex DO
  g_avoid_status[i] := 0;
END_FOR;

(* --- Clear all transporter states --- *)
FOR i := 1 TO MAX_Transporters DO
  g_transporter[i].IsActive          := FALSE;
  g_transporter[i].Status          := 0;
  g_transporter[i].Phase           := 0;
  g_transporter[i].TaskId         := 0;
  g_sim_trans[i].RunningTaskId := 0;
  g_transporter[i].LiftStationTarget    := 0;
  g_transporter[i].SinkStationTarget    := 0;
  g_sim_trans[i].TreatmentTime  := 0;
  g_sim_trans[i].LiftDeviceDelay := 0;
  g_sim_trans[i].SinkDeviceDelay := 0;
  g_transporter[i].DrippingTime   := 0;
  g_transporter[i].TaskRemainingTime  := 0;
  g_transporter[i].CurrentStation := 0;
  g_transporter[i].XFinalTarget  := 0;
  g_transporter[i].XDriveTarget  := 0;
  g_transporter[i].YFinalTarget  := 0;
  g_transporter[i].YDriveTarget  := 0;
  g_transporter[i].XPosition            := 0;
  g_transporter[i].YPosition            := 0;
  g_transporter[i].ZPosition            := 0;
  g_sim_trans[i].XVelocity           := 0;
  g_sim_trans[i].ZStage         := 0;
  g_sim_trans[i].ZTimer       := 0.0;
  g_transporter[i].XMinDriveLimit     := 0;
  g_transporter[i].XMaxDriveLimit     := 0;
END_FOR;

(* --- Clear all units --- *)
FOR i := 1 TO MAX_Units DO
  g_unit[i].location := 0;
  g_unit[i].Status   := 0;
  g_unit[i].Target   := 0;
END_FOR;

(* --- Clear NTT destinations --- *)
FOR i := 1 TO MAX_Transporters DO
  FOR j := 1 TO 8 DO
    g_ntt[i].Target[j].StationCount := 0;
    g_ntt[i].Target[j].FallbackCount := 0;
    FOR k := 1 TO MAX_STATIONS_PER_STEP DO
      g_ntt[i].Target[j].Stations[k] := 0;
      g_ntt[i].Target[j].FallbackStations[k] := 0;
    END_FOR;
  END_FOR;
END_FOR;

(* --- Clear all batches --- *)
FOR i := 1 TO MAX_Units DO
  g_batch[i].BatchCode  := 0;
  g_batch[i].State       := 0;
  g_batch[i].ProgId     := 0;
  g_batch[i].CurStage   := 0;
  g_batch[i].MinTime    := 0;
  g_batch[i].MaxTime    := 0;
  g_batch[i].CalTime    := 0;
  g_batch[i].StartTime  := LINT#0;
END_FOR;

(* --- Clear all treatment programs --- *)
FOR i := 1 TO MAX_Units DO
  g_program[i].ProgramId := 0;
  g_program[i].ProgramName := '';
  g_program[i].StepCount := 0;
  FOR j := 0 TO 30 DO
    FOR k := 0 TO 4 DO
      g_program[i].Steps[j].Stations[k] := 0;
    END_FOR;
    g_program[i].Steps[j].StationCount := 0;
    g_program[i].Steps[j].MinTime := 0;
    g_program[i].Steps[j].MaxTime := 0;
    g_program[i].Steps[j].CalTime := 0;
  END_FOR;
END_FOR;

(* --- Clear all schedules (g_schedule) --- *)
FOR i := 1 TO MAX_Units DO
  g_schedule[i].StageCount := 0;
  FOR j := 1 TO 30 DO
    g_schedule[i].Stages[j].station       := 0;
    g_schedule[i].Stages[j].EntryTime    := 0;
    g_schedule[i].Stages[j].ExitTime     := 0;
    g_schedule[i].Stages[j].MinTime      := 0;
    g_schedule[i].Stages[j].CalcTime     := 0;
    g_schedule[i].Stages[j].MaxTime      := 0;
    g_schedule[i].Stages[j].TransferTime := 0;
  END_FOR;
END_FOR;

(* --- Clear all task queues (g_task) --- *)
FOR i := 1 TO MAX_Transporters DO
  g_task[i].Count := 0;
  FOR j := 1 TO 60 DO
    g_task[i].Queue[j].Unit         := 0;
    g_task[i].Queue[j].Stage        := 0;
    g_task[i].Queue[j].LiftStationTarget := 0;
    g_task[i].Queue[j].SinkStationTarget := 0;
    g_task[i].Queue[j].StartTime   := 0;
    g_task[i].Queue[j].FinishTime  := 0;
    g_task[i].Queue[j].CalcTime    := 0;
    g_task[i].Queue[j].MinTime     := 0;
    g_task[i].Queue[j].MaxTime     := 0;
  END_FOR;
END_FOR;

(* --- Clear departure sandbox and pending write --- *)
g_dep_sandbox.Valid := FALSE;
g_dep_pending.Valid := FALSE;
g_dep_pending.BatchUnit  := 0;
g_dep_pending.BatchStage := 0;
g_dep_pending.BatchState := 0;

(* --- Clear departure scheduler state (previously missing) --- *)
g_dep_activated     := FALSE;
g_tsk_stable        := TRUE;   (* JS: tasksStableFlag starts true on empty line *)
g_dep_waiting_count := 0;
g_dep_wait_unit     := 0;
FOR i := 1 TO 5 DO
  g_dep_waiting[i] := 0;
END_FOR;

END_FUNCTION_BLOCK

(* ---- SIM_FB_EventQueue.st ---- *)
(* ============================================================
   SIM_FB_EventQueue — Event message queue handler (OPC UA)
   ============================================================
   Manages a circular 10-slot event queue (g_event).

   - enqueue: caller writes msg fields to g_event_pending,
     then sets g_event_pending_valid := TRUE.
     This FB picks it up and adds to queue.
   - dequeue: Gateway reads g_event.Buffer[Head] directly
     via OPC UA, then writes g_event_ack_seq to acknowledge.
     PLC sees ack match → advance head, count--.

   Called every PLC scan from plc_prg (always, not gated by
   scheduler turn).

   OPC UA handshake:
     PLC:    g_event.Count, g_event.Head, g_event.Buffer[] → readable via OPC UA
     Gateway: g_event_ack_seq → writable via OPC UA
     When g_event_ack_seq = g_event.Buffer[Head].Seq: message consumed → next.
   ============================================================ *)

FUNCTION_BLOCK SIM_FB_EventQueue
VAR_EXTERNAL
  g_event               : UDT_JC_EventQueueType;
  g_event_pending       : UDT_JC_EventMsgType;
  g_event_pending_valid : BOOL;
  g_event_ack_seq       : INT;
END_VAR
VAR
  tail : INT;
END_VAR

(* ── 1. Enqueue: pick up pending message if queue not full ── *)
IF g_event_pending_valid AND g_event.Count < 10 THEN
  tail := ((g_event.Head - 1 + g_event.Count) MOD 10) + 1;

  g_event_pending.Seq := g_event.NextSeq;
  g_event.NextSeq := g_event.NextSeq + 1;
  IF g_event.NextSeq > 32000 THEN
    g_event.NextSeq := 1;
  END_IF;

  g_event.Buffer[tail] := g_event_pending;
  g_event.Count := g_event.Count + 1;

  g_event_pending_valid := FALSE;
END_IF;

(* ── 2. Dequeue: check gateway ack for head message ── *)
IF g_event.Count > 0 THEN
  IF g_event_ack_seq = g_event.Buffer[g_event.Head].Seq THEN
    g_event.Head := (g_event.Head MOD 10) + 1;
    g_event.Count := g_event.Count - 1;
  END_IF;
END_IF;

END_FUNCTION_BLOCK

(* ---- SIM_FB_RunTasks.st ---- *)
(* ============================================================
   SIM_FB_RunTasks.st — Simulate transporter task execution

   For each active transporter [1..3], checks whether a new task
   has been assigned (task_id <> running_task_id) and executes
   the full transport cycle:

     Phase 0  idle        — waiting for new task
     Phase 1  to_lift     — X-drive towards lift station
     Phase 2  lifting     — Z-lift sequence (stages 1-5)
     Phase 3  to_sink     — X-drive towards sink station
     Phase 4  sinking     — Z-sink sequence (stages 6-8)

   Also maintains current_station (nearest station) every cycle.

   Called once per PLC scan from PLC_PRG.
   ============================================================ *)

FUNCTION_BLOCK SIM_FB_RunTasks
VAR_INPUT
  i_run : BOOL;       (* enable — typically init_done *)
END_VAR
VAR_EXTERNAL CONSTANT
    MAX_Transporters    : INT;
    MAX_Units           : INT;
    MAX_STEPS_PER_PROGRAM          : INT;
    MIN_StationIndex : INT;
    MAX_StationIndex   : INT;
    IN_PROCESS          : INT;
END_VAR

VAR_EXTERNAL
  g_transporter  : ARRAY[1..MAX_Transporters] OF UDT_TransporterStatusType;
  g_sim_trans    : ARRAY[1..MAX_Transporters] OF UDT_JC_SimTransporterType;
  g_station     : ARRAY[MIN_StationIndex..MAX_StationIndex] OF UDT_StationType;    g_station_loc  : ARRAY[1..MAX_StationIndex] OF UDT_UnitLocation;  g_cfg          : ARRAY[1..MAX_Transporters] OF UDT_TransporterType;
  g_move         : ARRAY[1..MAX_Transporters] OF UDT_JC_MoveTimesType;
  g_actual_move  : ARRAY[1..MAX_Transporters] OF UDT_JC_ActualMoveTimeType;
  g_unit         : ARRAY[1..MAX_Units] OF UDT_UnitType;
  g_batch        : ARRAY[1..MAX_Units] OF UDT_BatchType;
  g_program      : ARRAY[1..MAX_Units] OF UDT_TreatmentProgramType;
  g_time_s       : LINT;
  g_event_pending       : UDT_JC_EventMsgType;
  g_event_pending_valid : BOOL;
END_VAR
VAR
  i            : INT;
  idx          : INT;
  (* Physics FB instances — one per transporter (MATIEC needs separate instances) *)
  fb_x1        : SIM_FB_XMotion;
  fb_x2        : SIM_FB_XMotion;
  fb_x3        : SIM_FB_XMotion;
  fb_z1        : SIM_FB_ZMotion;
  fb_z2        : SIM_FB_ZMotion;
  fb_z3        : SIM_FB_ZMotion;
  (* Station lookup — now FC STC_FindStation, no instance needed *)
  (* Temp vars for VAR_IN_OUT passing *)
  tmp_x        : DINT;
  tmp_vx       : DINT;
  tmp_z        : DINT;
  tmp_zs       : INT;
  tmp_zt       : REAL;
  arrived_x    : BOOL;
  at_station   : BOOL;    (* TRUE only when actually at station, not just at drive limit *)
  arrived_z    : BOOL;
  station_kind : INT;
  device_delay : REAL;
  drop_time    : REAL;
  pick_unit_id : INT;     (* unit_id picked up from lift station *)
  xfer_total   : REAL;    (* transfer time for UI progress bar *)
  sink_unit_id : INT;     (* unit_id being placed at sink station *)
  (* Nearest-station calculation *)
  nearest_num  : INT;
  min_dist     : DINT;
  dx           : DINT;
  (* Actual move time tracker — now FC STC_TrackMoveTimes, no instance needed *)
  (* Unit location update — now FC STC_UpdateUnitLocation, no instance needed *)
  (* Event helpers *)
  evt_unit     : INT;
  evt_diff     : LINT;
  (* Treatment time wait *)
  can_lift       : BOOL;
  lift_uid       : INT;      (* unit at lift station *)
  treat_cal      : DINT;      (* treatment cal_time for current stage *)
  treat_elapsed  : LINT;     (* seconds spent at lift station *)
  (* ── TASK_COMPLETE event: phase timestamps per transporter ── *)
  ts_task_start  : ARRAY[1..3] OF LINT;  (* Phase 0→1: task accepted *)
  ts_at_lift     : ARRAY[1..3] OF LINT;  (* Phase 1 at_station: arrived at lift *)
  ts_lift_begin  : ARRAY[1..3] OF LINT;  (* Phase 1→2: can_lift, begin lift *)
  ts_lift_done   : ARRAY[1..3] OF LINT;  (* Phase 2→3: lift complete *)
  ts_at_sink     : ARRAY[1..3] OF LINT;  (* Phase 3→4: arrived at sink *)
  (* TASK_COMPLETE temp vars *)
  dd_lift_s      : INT;   (* lift device_delay in seconds *)
  dropping_s     : INT;   (* dropping/valutus time in seconds *)
  trip_s         : INT;   (* drip tray delay in seconds, 0 if not used *)
  dur_nosto      : INT;   (* computed nosto duration *)
  dur_lasku      : INT;   (* computed lasku duration *)
END_VAR

IF NOT i_run THEN
  RETURN;
END_IF;

FOR i := 1 TO MAX_Transporters DO
  IF g_transporter[i].IsActive THEN

  (* ── Phase 0 → 1: Accept new task ───────────────────────── *)
  IF (g_transporter[i].Phase = 0)
     AND (g_transporter[i].TaskId <> g_sim_trans[i].RunningTaskId) THEN
    g_sim_trans[i].RunningTaskId := g_transporter[i].TaskId;
    g_transporter[i].XFinalTarget := STC_FindStation(station_number := g_transporter[i].LiftStationTarget);
    g_transporter[i].Phase := 1;
    STC_TrackMoveTimes(i_trans := i, i_prev := 0, i_new := 1);
    g_transporter[i].Status := 4;  (* auto_run *)
    g_sim_trans[i].ZStage := 0;
    g_sim_trans[i].ZTimer := 0.0;
    (* Record task start timestamp *)
    ts_task_start[i] := g_time_s;
    ts_at_lift[i]    := LINT#0;

  (* ── Phase 1: Drive X towards lift station ──────────────── *)
  ELSIF g_transporter[i].Phase = 1 THEN
    tmp_x  := g_transporter[i].XPosition;
    tmp_vx := g_sim_trans[i].XVelocity;
    IF i = 1 THEN
      fb_x1(
        delta_t  := 0.02,
        x_target := g_transporter[i].XFinalTarget,
        x_min    := g_transporter[i].XMinDriveLimit,
        x_max    := g_transporter[i].XMaxDriveLimit,
        v_max    := g_cfg[i].SpeedMax_X,
        t_acc    := g_cfg[i].Acceleration_X,
        t_dec    := g_cfg[i].Deceleration_X,
        x_pos    := tmp_x,
        v_x      := tmp_vx
      );
      arrived_x := fb_x1.arrived;
    ELSIF i = 2 THEN
      fb_x2(
        delta_t  := 0.02,
        x_target := g_transporter[i].XFinalTarget,
        x_min    := g_transporter[i].XMinDriveLimit,
        x_max    := g_transporter[i].XMaxDriveLimit,
        v_max    := g_cfg[i].SpeedMax_X,
        t_acc    := g_cfg[i].Acceleration_X,
        t_dec    := g_cfg[i].Deceleration_X,
        x_pos    := tmp_x,
        v_x      := tmp_vx
      );
      arrived_x := fb_x2.arrived;
    ELSIF i = 3 THEN
      fb_x3(
        delta_t  := 0.02,
        x_target := g_transporter[i].XFinalTarget,
        x_min    := g_transporter[i].XMinDriveLimit,
        x_max    := g_transporter[i].XMaxDriveLimit,
        v_max    := g_cfg[i].SpeedMax_X,
        t_acc    := g_cfg[i].Acceleration_X,
        t_dec    := g_cfg[i].Deceleration_X,
        x_pos    := tmp_x,
        v_x      := tmp_vx
      );
      arrived_x := fb_x3.arrived;
    END_IF;
    g_transporter[i].XPosition  := tmp_x;
    g_sim_trans[i].XVelocity := tmp_vx;

    (* Only transition when actually at station, not just at drive limit *)
    at_station := arrived_x
                  AND (ABS(g_transporter[i].XPosition - g_transporter[i].XFinalTarget) <= 6);
    IF at_station THEN
      g_transporter[i].CurrentStation := g_transporter[i].LiftStationTarget;
      (* Record arrival at lift station (first time only) *)
      IF ts_at_lift[i] = LINT#0 THEN
        ts_at_lift[i] := g_time_s;
      END_IF;

      (* ── Wait for treatment time AND device_delay before lifting ──
         Z-movement starts when the LONGER of two has elapsed:
         1. Remaining treatment time (unit must finish treatment)
         2. Station device_delay (covers must be open)
         Both timers run simultaneously from transporter arrival.
         This matches JS behavior: max(treatment, device_delay). *)
      can_lift := TRUE;
      STC_FindStation(station_number := g_transporter[i].LiftStationTarget, device_delay_s => device_delay, dropping_time_s => drop_time);

      (* Check treatment time *)
      lift_uid := g_station_loc[g_transporter[i].LiftStationTarget].UnitId;
      IF lift_uid >= 1 AND lift_uid <= MAX_Units THEN
        IF g_batch[lift_uid].State = IN_PROCESS
           AND g_batch[lift_uid].CurStage >= 1
           AND g_batch[lift_uid].CurStage <= MAX_STEPS_PER_PROGRAM THEN
          treat_cal := g_program[lift_uid].Steps[g_batch[lift_uid].CurStage].CalTime;
          IF treat_cal > 0 THEN
            treat_elapsed := g_time_s - g_station_loc[g_transporter[i].LiftStationTarget].ChangeTime;
            IF treat_elapsed < DINT_TO_LINT(treat_cal) THEN
              can_lift := FALSE;
            END_IF;
          END_IF;
        END_IF;
      END_IF;

      (* Check device_delay — covers must have had time to open since arrival *)
      IF can_lift AND device_delay > 0.0 THEN
        IF LINT_TO_REAL(g_time_s - ts_at_lift[i]) < device_delay THEN
          can_lift := FALSE;
        END_IF;
      END_IF;

      IF can_lift THEN
      (* Record lift begin timestamp *)
      ts_lift_begin[i] := g_time_s;
      (* drop_time already captured by STC_FindStation above *)
      (* Skip stage 1 — device_delay already overlapped above.
         Z-movement starts immediately (stage 2).
         dropping_time and drip_tray_delay happen at the TOP. *)
      g_transporter[i].ZPosition := 0;
      g_sim_trans[i].ZTimer := 0.0;
      g_sim_trans[i].ZStage := 2;
      g_transporter[i].Phase := 2;
      STC_TrackMoveTimes(i_trans := i, i_prev := 1, i_new := 2);

      (* ── Calculate transfer time (used by event + batch times) ── *)
      xfer_total := STC_CalcTransferTime(
        i_from_stn            := g_transporter[i].LiftStationTarget,
        i_to_stn              := g_transporter[i].SinkStationTarget,
        i_move                := g_move[i],
        i_from_dropping_x10   := g_station[g_transporter[i].LiftStationTarget].DrippingTime,
        i_to_device_delay_x10 := g_station[g_transporter[i].SinkStationTarget].DeviceDelay,
        i_drip_tray_delay_x10 := g_cfg[i].DripTrayDelay
      );
      IF xfer_total < 1.0 THEN
        xfer_total := INT_TO_REAL(
          ABS(g_transporter[i].SinkStationTarget
              - g_transporter[i].LiftStationTarget)
        ) * 8.0;
      END_IF;
      IF xfer_total < 5.0 THEN xfer_total := 60.0; END_IF;

      (* ── Emit LIFT event (msg_type=2) ── *)
      evt_unit := g_station_loc[g_transporter[i].LiftStationTarget].UnitId;
      IF NOT g_event_pending_valid AND evt_unit >= 1 THEN
        g_event_pending.MsgType := 2;
        g_event_pending.TsHi := LINT_TO_INT(g_time_s / LINT#65536);
        g_event_pending.TsLo := LINT_TO_INT(g_time_s MOD LINT#65536);
        g_event_pending.Payload[1]  := LINT_TO_INT(g_transporter[i].TaskId / LINT#65536);   (* TaskId_Hi *)
        g_event_pending.Payload[2]  := LINT_TO_INT(g_transporter[i].TaskId MOD LINT#65536);  (* TaskId_Lo *)
        g_event_pending.Payload[3]  := i;
        g_event_pending.Payload[4]  := evt_unit;
        g_event_pending.Payload[5]  := g_transporter[i].LiftStationTarget;
        g_event_pending.Payload[6]  := g_batch[evt_unit].BatchCode;
        g_event_pending.Payload[7]  := g_batch[evt_unit].CurStage;
        evt_diff := g_time_s - g_station_loc[g_transporter[i].LiftStationTarget].ChangeTime;
        IF evt_diff > LINT#32000 THEN
          g_event_pending.Payload[8] := 32000;
        ELSE
          g_event_pending.Payload[8] := LINT_TO_INT(evt_diff);
        END_IF;
        (* ── Original program calc/min/max for this stage ── *)
        (* g_sim_trans holds dispatch-time scheduler values which may differ
           from the treatment program originals. Read directly from g_program
           using the batch's current stage (CurStage=1-based program index). *)
        IF g_batch[evt_unit].CurStage >= 1 AND g_batch[evt_unit].CurStage <= 30 THEN
          g_event_pending.Payload[9]  := DINT_TO_INT(g_program[evt_unit].Steps[g_batch[evt_unit].CurStage].CalTime);
          g_event_pending.Payload[10] := DINT_TO_INT(g_program[evt_unit].Steps[g_batch[evt_unit].CurStage].MinTime);
          g_event_pending.Payload[11] := DINT_TO_INT(g_program[evt_unit].Steps[g_batch[evt_unit].CurStage].MaxTime);
        ELSE
          (* Stage 0 (pickup) — no program step *)
          g_event_pending.Payload[9]  := 0;
          g_event_pending.Payload[10] := 0;
          g_event_pending.Payload[11] := 0;
        END_IF;
        g_event_pending.Payload[12] := REAL_TO_INT(xfer_total);
        g_event_pending_valid := TRUE;
      END_IF;

      (* Unit moves from lift station → transporter *)
      pick_unit_id := g_station_loc[g_transporter[i].LiftStationTarget].UnitId;
      IF pick_unit_id >= 1 THEN
        STC_UpdateUnitLocation(i_unit := pick_unit_id, i_location := i);

        (* Set batch transfer times for UI progress bar — matches JS behavior *)
        g_batch[pick_unit_id].StartTime := g_time_s;
        g_batch[pick_unit_id].CalTime   := REAL_TO_DINT(xfer_total);
        g_batch[pick_unit_id].MinTime   := g_batch[pick_unit_id].CalTime;
        g_batch[pick_unit_id].MaxTime   := 600;
      END_IF;
      END_IF;  (* can_lift *)
    END_IF;
    (* If arrived_x but not at_station → at drive limit, wait for clearance *)

  (* ── Phase 2: Lift Z at lift station ────────────────────── *)
  ELSIF g_transporter[i].Phase = 2 THEN
    STC_FindStation(station_number := g_transporter[i].LiftStationTarget, skind => station_kind);
    tmp_z  := g_transporter[i].ZPosition;
    tmp_zs := g_sim_trans[i].ZStage;
    tmp_zt := g_sim_trans[i].ZTimer;
    IF i = 1 THEN
      fb_z1(
        delta_t       := 0.02,
        station_kind  := station_kind,
        ZPosDown        := g_cfg[i].ZPosDown,
        ZPosUp          := 0,
        ZPosSlowUp      := g_cfg[i].ZPosSlowUp,
        ZPosSlowDown    := g_cfg[i].ZPosSlowDown,
        ZPosSlowEnd     := g_cfg[i].ZPosSlowEnd,
        SpeedLiftSlow_Z := g_cfg[i].SpeedLiftSlow_Z,
        SpeedLiftFast_Z := g_cfg[i].SpeedLiftFast_Z,
        DripTrayDelay   := g_cfg[i].DripTrayDelay,
        DroppingTime    := g_station[g_transporter[i].LiftStationTarget].DrippingTime,
        z_mm          := tmp_z,
        z_stage       := tmp_zs,
        z_timer_s     := tmp_zt
      );
      arrived_z := fb_z1.done;
    ELSIF i = 2 THEN
      fb_z2(
        delta_t       := 0.02,
        station_kind  := station_kind,
        ZPosDown        := g_cfg[i].ZPosDown,
        ZPosUp          := 0,
        ZPosSlowUp      := g_cfg[i].ZPosSlowUp,
        ZPosSlowDown    := g_cfg[i].ZPosSlowDown,
        ZPosSlowEnd     := g_cfg[i].ZPosSlowEnd,
        SpeedLiftSlow_Z := g_cfg[i].SpeedLiftSlow_Z,
        SpeedLiftFast_Z := g_cfg[i].SpeedLiftFast_Z,
        DripTrayDelay   := g_cfg[i].DripTrayDelay,
        DroppingTime    := g_station[g_transporter[i].LiftStationTarget].DrippingTime,
        z_mm          := tmp_z,
        z_stage       := tmp_zs,
        z_timer_s     := tmp_zt
      );
      arrived_z := fb_z2.done;
    ELSIF i = 3 THEN
      fb_z3(
        delta_t       := 0.02,
        station_kind  := station_kind,
        ZPosDown        := g_cfg[i].ZPosDown,
        ZPosUp          := 0,
        ZPosSlowUp      := g_cfg[i].ZPosSlowUp,
        ZPosSlowDown    := g_cfg[i].ZPosSlowDown,
        ZPosSlowEnd     := g_cfg[i].ZPosSlowEnd,
        SpeedLiftSlow_Z := g_cfg[i].SpeedLiftSlow_Z,
        SpeedLiftFast_Z := g_cfg[i].SpeedLiftFast_Z,
        DripTrayDelay   := g_cfg[i].DripTrayDelay,
        DroppingTime    := g_station[g_transporter[i].LiftStationTarget].DrippingTime,
        z_mm          := tmp_z,
        z_stage       := tmp_zs,
        z_timer_s     := tmp_zt
      );
      arrived_z := fb_z3.done;
    END_IF;
    g_transporter[i].ZPosition      := tmp_z;
    g_sim_trans[i].ZStage   := tmp_zs;
    g_sim_trans[i].ZTimer := tmp_zt;
    IF arrived_z THEN
      (* Record lift done timestamp *)
      ts_lift_done[i] := g_time_s;
      g_transporter[i].XFinalTarget := STC_FindStation(station_number := g_transporter[i].SinkStationTarget);
      g_transporter[i].Phase := 3;
      STC_TrackMoveTimes(i_trans := i, i_prev := 2, i_new := 3);
    END_IF;

  (* ── Phase 3: Drive X towards sink station ─────────────── *)
  ELSIF g_transporter[i].Phase = 3 THEN
    tmp_x  := g_transporter[i].XPosition;
    tmp_vx := g_sim_trans[i].XVelocity;
    IF i = 1 THEN
      fb_x1(
        delta_t  := 0.02,
        x_target := g_transporter[i].XFinalTarget,
        x_min    := g_transporter[i].XMinDriveLimit,
        x_max    := g_transporter[i].XMaxDriveLimit,
        v_max    := g_cfg[i].SpeedMax_X,
        t_acc    := g_cfg[i].Acceleration_X,
        t_dec    := g_cfg[i].Deceleration_X,
        x_pos    := tmp_x,
        v_x      := tmp_vx
      );
      arrived_x := fb_x1.arrived;
    ELSIF i = 2 THEN
      fb_x2(
        delta_t  := 0.02,
        x_target := g_transporter[i].XFinalTarget,
        x_min    := g_transporter[i].XMinDriveLimit,
        x_max    := g_transporter[i].XMaxDriveLimit,
        v_max    := g_cfg[i].SpeedMax_X,
        t_acc    := g_cfg[i].Acceleration_X,
        t_dec    := g_cfg[i].Deceleration_X,
        x_pos    := tmp_x,
        v_x      := tmp_vx
      );
      arrived_x := fb_x2.arrived;
    ELSIF i = 3 THEN
      fb_x3(
        delta_t  := 0.02,
        x_target := g_transporter[i].XFinalTarget,
        x_min    := g_transporter[i].XMinDriveLimit,
        x_max    := g_transporter[i].XMaxDriveLimit,
        v_max    := g_cfg[i].SpeedMax_X,
        t_acc    := g_cfg[i].Acceleration_X,
        t_dec    := g_cfg[i].Deceleration_X,
        x_pos    := tmp_x,
        v_x      := tmp_vx
      );
      arrived_x := fb_x3.arrived;
    END_IF;
    g_transporter[i].XPosition  := tmp_x;
    g_sim_trans[i].XVelocity := tmp_vx;

    (* Only transition when actually at station, not just at drive limit *)
    at_station := arrived_x
                  AND (ABS(g_transporter[i].XPosition - g_transporter[i].XFinalTarget) <= 6);
    IF at_station THEN
      g_transporter[i].CurrentStation := g_transporter[i].SinkStationTarget;
      (* Record arrival at sink timestamp *)
      ts_at_sink[i] := g_time_s;
      STC_FindStation(station_number := g_transporter[i].SinkStationTarget, device_delay_s => device_delay);
      g_sim_trans[i].ZTimer := device_delay + INT_TO_REAL(g_cfg[i].DripTrayDelay) / 10.0;
      g_sim_trans[i].ZStage := 6;
      g_transporter[i].Phase := 4;
      STC_TrackMoveTimes(i_trans := i, i_prev := 3, i_new := 4);
    END_IF;
    (* If arrived_x but not at_station → at drive limit, wait for clearance *)

  (* ── Phase 4: Sink Z at sink station ───────────────────── *)
  ELSIF g_transporter[i].Phase = 4 THEN
    STC_FindStation(station_number := g_transporter[i].SinkStationTarget, skind => station_kind);
    tmp_z  := g_transporter[i].ZPosition;
    tmp_zs := g_sim_trans[i].ZStage;
    tmp_zt := g_sim_trans[i].ZTimer;
    IF i = 1 THEN
      fb_z1(
        delta_t       := 0.02,
        station_kind  := station_kind,
        ZPosDown        := g_cfg[i].ZPosDown,
        ZPosUp          := 0,
        ZPosSlowUp      := g_cfg[i].ZPosSlowUp,
        ZPosSlowDown    := g_cfg[i].ZPosSlowDown,
        ZPosSlowEnd     := g_cfg[i].ZPosSlowEnd,
        SpeedLiftSlow_Z := g_cfg[i].SpeedLiftSlow_Z,
        SpeedLiftFast_Z := g_cfg[i].SpeedLiftFast_Z,
        DripTrayDelay   := g_cfg[i].DripTrayDelay,
        DroppingTime    := 0,
        z_mm          := tmp_z,
        z_stage       := tmp_zs,
        z_timer_s     := tmp_zt
      );
      arrived_z := fb_z1.done;
    ELSIF i = 2 THEN
      fb_z2(
        delta_t       := 0.02,
        station_kind  := station_kind,
        ZPosDown        := g_cfg[i].ZPosDown,
        ZPosUp          := 0,
        ZPosSlowUp      := g_cfg[i].ZPosSlowUp,
        ZPosSlowDown    := g_cfg[i].ZPosSlowDown,
        ZPosSlowEnd     := g_cfg[i].ZPosSlowEnd,
        SpeedLiftSlow_Z := g_cfg[i].SpeedLiftSlow_Z,
        SpeedLiftFast_Z := g_cfg[i].SpeedLiftFast_Z,
        DripTrayDelay   := g_cfg[i].DripTrayDelay,
        DroppingTime    := 0,
        z_mm          := tmp_z,
        z_stage       := tmp_zs,
        z_timer_s     := tmp_zt
      );
      arrived_z := fb_z2.done;
    ELSIF i = 3 THEN
      fb_z3(
        delta_t       := 0.02,
        station_kind  := station_kind,
        ZPosDown        := g_cfg[i].ZPosDown,
        ZPosUp          := 0,
        ZPosSlowUp      := g_cfg[i].ZPosSlowUp,
        ZPosSlowDown    := g_cfg[i].ZPosSlowDown,
        ZPosSlowEnd     := g_cfg[i].ZPosSlowEnd,
        SpeedLiftSlow_Z := g_cfg[i].SpeedLiftSlow_Z,
        SpeedLiftFast_Z := g_cfg[i].SpeedLiftFast_Z,
        DripTrayDelay   := g_cfg[i].DripTrayDelay,
        DroppingTime    := 0,
        z_mm          := tmp_z,
        z_stage       := tmp_zs,
        z_timer_s     := tmp_zt
      );
      arrived_z := fb_z3.done;
    END_IF;
    g_transporter[i].ZPosition      := tmp_z;
    g_sim_trans[i].ZStage   := tmp_zs;
    g_sim_trans[i].ZTimer := tmp_zt;
    IF arrived_z THEN
      (* ── Emit TASK_COMPLETE event (msg_type=3) before Phase reset ── *)
      IF NOT g_event_pending_valid THEN
        (* Config-based sub-phase durations *)
        dropping_s := g_transporter[i].DrippingTime / 10;
        IF g_cfg[i].DripTrayInUse THEN
          trip_s := g_cfg[i].DripTrayDelay / 10;
        ELSE
          trip_s := 0;
        END_IF;
        (* Nosto = total lift phase - dropping - trip_close
           device_delay no longer in lift phase (overlapped in Phase 1) *)
        dur_nosto := LINT_TO_INT(ts_lift_done[i] - ts_lift_begin[i])
                     - dropping_s - trip_s;
        IF dur_nosto < 0 THEN dur_nosto := 0; END_IF;
        (* Lasku = total sink phase - device_delay - trip_open *)
        dd_lift_s := g_sim_trans[i].SinkDeviceDelay / 10;
        dur_lasku := LINT_TO_INT(g_time_s - ts_at_sink[i]) - dd_lift_s - trip_s;
        IF dur_lasku < 0 THEN dur_lasku := 0; END_IF;

        g_event_pending.MsgType := 3;
        g_event_pending.TsHi := LINT_TO_INT(g_time_s / LINT#65536);
        g_event_pending.TsLo := LINT_TO_INT(g_time_s MOD LINT#65536);
        g_event_pending.Payload[1]  := LINT_TO_INT(g_transporter[i].TaskId / LINT#65536);   (* TaskId_Hi *)
        g_event_pending.Payload[2]  := LINT_TO_INT(g_transporter[i].TaskId MOD LINT#65536);  (* TaskId_Lo *)
        g_event_pending.Payload[3]  := i;                                                     (* transporter *)
        g_event_pending.Payload[4]  := LINT_TO_INT(ts_at_lift[i] - ts_task_start[i]);         (* siirto nostoasemalle *)
        g_event_pending.Payload[5]  := LINT_TO_INT(ts_lift_begin[i] - ts_at_lift[i]);         (* odotus ennen nostoa (max(treat,dev_delay)) *)
        g_event_pending.Payload[6]  := dur_nosto;                                             (* nosto *)
        g_event_pending.Payload[7]  := dropping_s;                                            (* valutus *)
        g_event_pending.Payload[8]  := trip_s;                                                (* trip close *)
        g_event_pending.Payload[9]  := LINT_TO_INT(ts_at_sink[i] - ts_lift_done[i]);          (* siirto laskuasemalle *)
        g_event_pending.Payload[10] := trip_s;                                                (* trip open *)
        g_event_pending.Payload[11] := dur_lasku;                                             (* lasku *)
        g_event_pending.Payload[12] := LINT_TO_INT(g_time_s - ts_task_start[i]);              (* total *)
        g_event_pending_valid := TRUE;
      END_IF;

      (* Unit moves from transporter → sink station *)
      sink_unit_id := g_station_loc[i].UnitId;
      IF sink_unit_id >= 1 THEN
        STC_UpdateUnitLocation(i_unit := sink_unit_id, i_location := g_transporter[i].SinkStationTarget, i_ntt_primary := g_sim_trans[i].NttPrimary);
      END_IF;

      g_transporter[i].Phase := 0;
      STC_TrackMoveTimes(i_trans := i, i_prev := 4, i_new := 0);
      g_transporter[i].Status := 3;  (* auto_idle *)

    END_IF;
  END_IF;  (* ELSIF chain: phases 0→1→2→3→4 *)

  (* ── Phase 0 idle: drive back inside limits if outside ────── *)
  IF g_transporter[i].Phase = 0 THEN
    tmp_x  := g_transporter[i].XPosition;
    tmp_vx := g_sim_trans[i].XVelocity;
    (* Use current position as target — XMotion will clamp to nearest limit if outside *)
    IF i = 1 THEN
      fb_x1(
        delta_t  := 0.02,
        x_target := tmp_x,
        x_min    := g_transporter[i].XMinDriveLimit,
        x_max    := g_transporter[i].XMaxDriveLimit,
        v_max    := g_cfg[i].SpeedMax_X,
        t_acc    := g_cfg[i].Acceleration_X,
        t_dec    := g_cfg[i].Deceleration_X,
        x_pos    := tmp_x,
        v_x      := tmp_vx
      );
    ELSIF i = 2 THEN
      fb_x2(
        delta_t  := 0.02,
        x_target := tmp_x,
        x_min    := g_transporter[i].XMinDriveLimit,
        x_max    := g_transporter[i].XMaxDriveLimit,
        v_max    := g_cfg[i].SpeedMax_X,
        t_acc    := g_cfg[i].Acceleration_X,
        t_dec    := g_cfg[i].Deceleration_X,
        x_pos    := tmp_x,
        v_x      := tmp_vx
      );
    ELSIF i = 3 THEN
      fb_x3(
        delta_t  := 0.02,
        x_target := tmp_x,
        x_min    := g_transporter[i].XMinDriveLimit,
        x_max    := g_transporter[i].XMaxDriveLimit,
        v_max    := g_cfg[i].SpeedMax_X,
        t_acc    := g_cfg[i].Acceleration_X,
        t_dec    := g_cfg[i].Deceleration_X,
        x_pos    := tmp_x,
        v_x      := tmp_vx
      );
    END_IF;
    g_transporter[i].XPosition  := tmp_x;
    g_sim_trans[i].XVelocity := tmp_vx;
  END_IF;

  (* ── Nearest station tracking ──────────────────────────── *)
  min_dist := 999999999;
  nearest_num := g_transporter[i].CurrentStation;
  FOR idx := MIN_StationIndex TO MAX_StationIndex DO
    IF g_station[idx].TankId <> 0 THEN
      dx := g_station[idx].XPosition - g_transporter[i].XPosition;
      IF ABS(dx) < min_dist THEN
        min_dist := ABS(dx);
        nearest_num := idx;
      END_IF;
    END_IF;
  END_FOR;
  g_transporter[i].CurrentStation := nearest_num;

  END_IF;  (* active *)
END_FOR;

END_FUNCTION_BLOCK

(* ---- SIM_FB_XMotion.st ---- *)
(* ============================================================
   SIM_FB_XMotion — Horizontal motion with accel / decel

   Company : Galvatek part of the John Cockerill Group
   Author  : Jarmo Piipponen
   Created : 25.03.2026
   ============================================================
   Trapezoidal velocity profile: accelerate, cruise, decelerate.
   Clamps position to [x_min..x_max] drive limits.
   VAR_IN_OUT: x_pos, v_x (modified in place).
   ------------------------------------------------------------
   Changes:
   ============================================================ *)

FUNCTION_BLOCK SIM_FB_XMotion
VAR_INPUT
  delta_t  : REAL;     (* cycle time s — simulation internal *)
  x_target : DINT;     (* target X mm *)
  x_min    : DINT;     (* TWA lower limit mm *)
  x_max    : DINT;     (* TWA upper limit mm *)
  v_max    : DINT;     (* max velocity mm/s *)
  t_acc    : DINT;     (* acceleration time ×10 = tenths of second *)
  t_dec    : DINT;     (* deceleration time ×10 = tenths of second *)
END_VAR
VAR_IN_OUT
  x_pos : DINT;        (* current X position mm *)
  v_x   : DINT;        (* current X velocity mm/s *)
END_VAR
VAR_OUTPUT
  arrived : BOOL;
END_VAR
VAR
  (* Internal REAL copies for physics integration *)
  r_target     : REAL;
  r_min        : REAL;
  r_max        : REAL;
  r_vmax       : REAL;
  r_tacc       : REAL;
  r_tdec       : REAL;
  r_pos        : REAL;
  r_vel        : REAL;
  drive_target : REAL;
  distance     : REAL;
  dir          : REAL;
  a_acc        : REAL;
  a_dec        : REAL;
  brake_dist   : REAL;
  new_vel      : REAL;
  travel       : REAL;
END_VAR
  (* Convert DINT/INT inputs to REAL for physics *)
  r_target := DINT_TO_REAL(x_target);
  r_min    := DINT_TO_REAL(x_min);
  r_max    := DINT_TO_REAL(x_max);
  r_vmax   := DINT_TO_REAL(v_max);
  r_tacc   := DINT_TO_REAL(t_acc) / 10.0;
  r_tdec   := DINT_TO_REAL(t_dec) / 10.0;
  r_pos    := DINT_TO_REAL(x_pos);
  r_vel    := DINT_TO_REAL(v_x);

  IF (r_max > r_min) THEN
    IF r_pos < r_min THEN
      drive_target := r_min;
    ELSIF r_pos > r_max THEN
      drive_target := r_max;
    ELSE
      IF r_target < r_min THEN
        drive_target := r_min;
      ELSIF r_target > r_max THEN
        drive_target := r_max;
      ELSE
        drive_target := r_target;
      END_IF;
    END_IF;
  ELSE
    drive_target := r_target;
  END_IF;

  arrived := ABS(r_pos - drive_target) <= 3.0;
  IF arrived THEN
    x_pos := REAL_TO_DINT(drive_target);
    v_x := 0;
    RETURN;
  END_IF;

  IF r_tacc <= 0.0 THEN r_tacc := 0.001; END_IF;
  IF r_tdec <= 0.0 THEN r_tdec := 0.001; END_IF;
  IF r_vmax < 0.0 THEN r_vmax := 0.0; END_IF;

  a_acc := r_vmax / r_tacc;
  a_dec := r_vmax / r_tdec;

  dir := 1.0;
  IF drive_target < r_pos THEN
    dir := -1.0;
  END_IF;

  distance := ABS(drive_target - r_pos);

  IF a_dec > 0.0 THEN
    brake_dist := (r_vel * r_vel) / (2.0 * a_dec);
  ELSE
    brake_dist := 0.0;
  END_IF;

  IF brake_dist >= distance THEN
    new_vel := r_vel - a_dec * delta_t;
    IF new_vel < 0.0 THEN new_vel := 0.0; END_IF;
  ELSE
    new_vel := r_vel + a_acc * delta_t;
    IF new_vel > r_vmax THEN new_vel := r_vmax; END_IF;
  END_IF;

  travel := new_vel * delta_t;
  IF travel >= distance THEN
    x_pos := REAL_TO_DINT(drive_target);
    v_x := 0;
    arrived := TRUE;
  ELSE
    x_pos := REAL_TO_DINT(r_pos + dir * travel);
    v_x := REAL_TO_DINT(new_vel);
    arrived := FALSE;
  END_IF;
END_FUNCTION_BLOCK

(* ---- SIM_FB_ZMotion.st ---- *)
(* ============================================================
   SIM_FB_ZMotion.st — Vertical (Z) motion simulation

   Simulates 2D transporter lift/sink with realistic physics:
   - Slow start / fast middle / slow end speed profiles
   - Different slow zones for wet vs dry stations
   - Device delays and drip delays

   Coordinate convention: z=0 is bottom (sunk), z=z_total is top (lifted)

   LIFT sequence (z_stage 2-5, 9):
     2: Slow lift    0 → ZPosSlowUp/ZPosSlowDown
     3: Fast lift    → (z_total - ZPosSlowEnd)
     4: Slow end     → z_total
     5: Dropping     at top, dripping time (blue bar in UI)
     9: Drip close   drip tray close delay at top

   Note: Device delay + treatment overlap is handled by the caller
   (SIM_FB_RunTasks) in Phase 1 via can_lift check. Stage 1 is
   no longer used for lift — caller sets z_stage := 2 directly.

   SINK sequence (z_stage 6-8):
     6: Init delay  (device_delay + drip_delay)
     7: Fast sink    z_total → slow_zone
     8: Slow sink    → 0 mm

   Caller sets z_stage and z_timer_s before first call.
   Output 'done' pulses TRUE when sequence completes.
   ============================================================ *)

FUNCTION_BLOCK SIM_FB_ZMotion
VAR_INPUT
  delta_t         : REAL;    (* Cycle time in seconds — simulation internal *)
  station_kind    : INT;     (* KIND_DRY=0, KIND_WET=1 *)
  ZPosUp          : DINT;    (* Z position at full up mm *)
  ZPosDown        : DINT;    (* Z position at full down mm *)
  ZPosSlowUp      : DINT;    (* Slow zone when going up (dry) mm *)
  ZPosSlowDown    : DINT;    (* Slow zone when going down (wet) mm *)
  ZPosSlowEnd     : DINT;    (* Slow zone at end of travel mm *)
  SpeedLiftSlow_Z : DINT;    (* Slow speed mm/s *)
  SpeedLiftFast_Z : DINT;    (* Fast speed mm/s *)
  DripTrayDelay   : INT;     (* Drip tray open/close delay ×10 = tenths of second *)
  DroppingTime    : INT;     (* Dropping/dripping time ×10 = tenths of second *)
END_VAR
VAR_IN_OUT
  z_mm      : DINT;        (* Current Z position mm *)
  z_stage   : INT;         (* Current motion stage *)
  z_timer_s : REAL;        (* Delay timer — simulation internal *)
END_VAR
VAR_OUTPUT
  done : BOOL;             (* TRUE when sequence complete *)
END_VAR
VAR_EXTERNAL CONSTANT
  KIND_WET : INT;
END_VAR
VAR
  (* Internal REAL copies for physics integration *)
  r_z          : REAL;
  r_total      : REAL;
  r_slow_zone  : REAL;
  r_slow_end   : REAL;
  r_slow_spd   : REAL;
  r_fast_spd   : REAL;
  r_drip       : REAL;
  r_drop       : REAL;     (* dropping/dripping time seconds *)
  z_total_mm   : DINT;     (* computed: ZPosDown - ZPosUp *)
END_VAR

  done := FALSE;
  z_total_mm := ZPosDown - ZPosUp;

  (* Convert DINT/INT inputs to REAL for physics *)
  r_z         := DINT_TO_REAL(z_mm);
  r_total     := DINT_TO_REAL(z_total_mm);
  r_slow_end  := DINT_TO_REAL(ZPosSlowEnd);
  r_slow_spd  := DINT_TO_REAL(SpeedLiftSlow_Z);
  r_fast_spd  := DINT_TO_REAL(SpeedLiftFast_Z);
  r_drip      := INT_TO_REAL(DripTrayDelay) / 10.0;
  r_drop      := INT_TO_REAL(DroppingTime) / 10.0;

  (* Select slow zone based on station kind *)
  IF station_kind = KIND_WET THEN
    r_slow_zone := DINT_TO_REAL(ZPosSlowDown);
  ELSE
    r_slow_zone := DINT_TO_REAL(ZPosSlowUp);
  END_IF;

  CASE z_stage OF

    (* === LIFT: stages 2-5,9 — nosto altaasta ylös (z kasvaa: 0 → z_total) === *)
    (* Stage 1 no longer used for lift — device_delay overlaps with treatment wait *)

    2: (* Slow lift start — hidas nosto nesteestä *)
      r_z := r_z + r_slow_spd * delta_t;
      z_mm := REAL_TO_DINT(r_z);
      IF r_z >= r_slow_zone THEN
        z_stage := 3;
      END_IF;

    3: (* Fast lift — nopea nosto *)
      r_z := r_z + r_fast_spd * delta_t;
      z_mm := REAL_TO_DINT(r_z);
      IF r_z >= (r_total - r_slow_end) THEN
        z_stage := 4;
      END_IF;

    4: (* Slow lift end — hidas loppunosto *)
      r_z := r_z + r_slow_spd * delta_t;
      IF r_z >= r_total THEN
        z_mm := z_total_mm;
        z_timer_s := r_drop;
        z_stage := 5;
      ELSE
        z_mm := REAL_TO_DINT(r_z);
      END_IF;

    5: (* Dropping / dripping — valutusaika yläasemassa *)
      z_timer_s := z_timer_s - delta_t;
      IF z_timer_s <= 0.0 THEN
        z_timer_s := r_drip;
        z_stage := 9;
      END_IF;

    9: (* Drip tray close — tippakouru sulkeutuu *)
      z_timer_s := z_timer_s - delta_t;
      IF z_timer_s <= 0.0 THEN
        z_stage := 0;
        done := TRUE;
      END_IF;

    (* === SINK: stages 6-8 — lasku altaaseen (z pienenee: z_total → 0) === *)

    6: (* Init delay: device_delay + drip_delay *)
      z_timer_s := z_timer_s - delta_t;
      IF z_timer_s <= 0.0 THEN
        z_stage := 7;
      END_IF;

    7: (* Fast sink — nopea lasku *)
      r_z := r_z - r_fast_spd * delta_t;
      z_mm := REAL_TO_DINT(r_z);
      IF r_z <= r_slow_zone THEN
        z_stage := 8;
      END_IF;

    8: (* Slow sink — hidas lasku nesteeseen *)
      r_z := r_z - r_slow_spd * delta_t;
      IF r_z <= 0.0 THEN
        z_mm := 0;
        z_stage := 0;
        done := TRUE;
      ELSE
        z_mm := REAL_TO_DINT(r_z);
      END_IF;

  END_CASE;

END_FUNCTION_BLOCK

(* ---- STC_FB_CalcMoveTimes.st ---- *)
(* ============================================================
   STC_FB_CalcMoveTimes — Compute g_move from kinematic params
   ============================================================
   Calculates precomputed movement times for all active
   transporters using calibration kinematic parameters (g_cal)
   and station positions (g_station).

   For each transporter with valid g_cal data (x_max_mm_s > 0):
     - lift_s/sink_s: based on station kind (0=dry, 1=wet)
     - travel: trapezoidal velocity profile from X distances

   Call with i_run = TRUE to trigger computation (rising edge).

   Replaces need to re-run full calibration sequence when
   kinematic parameters are already known (e.g. loaded from
   a previously saved movement_times.json).
   ============================================================ *)

FUNCTION_BLOCK STC_FB_CalcMoveTimes
VAR_INPUT
  i_run : BOOL;    (* rising edge triggers computation *)
END_VAR
VAR_EXTERNAL CONSTANT
    MAX_Transporters    : INT;
    MIN_StationIndex : INT;
    MAX_StationIndex   : INT;
END_VAR
VAR_EXTERNAL
  g_cal           : ARRAY[1..MAX_Transporters] OF UDT_JC_CalibrationType;
  g_station       : ARRAY[MIN_StationIndex..MAX_StationIndex] OF UDT_StationType;
  g_move          : ARRAY[1..MAX_Transporters] OF UDT_JC_MoveTimesType;
  g_station_count : INT;
END_VAR
VAR
  prev_run  : BOOL := FALSE;
  tid       : INT;
  si        : INT;
  sj        : INT;
  idx_i     : INT;
  idx_j     : INT;
  last_stn  : INT;    (* last active station number *)
  vm        : REAL;   (* max velocity mm/s *)
  ta        : REAL;   (* accel time s *)
  td        : REAL;   (* decel time s *)
  d_acc     : REAL;   (* accel distance mm *)
  d_dec     : REAL;   (* decel distance mm *)
  dist      : REAL;   (* distance between stations mm *)
  t_time    : REAL;   (* computed travel time *)
  v_peak    : REAL;   (* peak velocity in triangle profile *)
END_VAR

(* Rising edge detection *)
IF i_run AND NOT prev_run THEN

  (* Determine last active station *)
  last_stn := MIN_StationIndex + g_station_count - 1;
  IF last_stn > MAX_StationIndex THEN
    last_stn := MAX_StationIndex;
  END_IF;

  FOR tid := 1 TO MAX_Transporters DO
    (* Skip transporters without valid calibration data *)
    IF g_cal[tid].XMaxSpeed >= 1 THEN

      vm := DINT_TO_REAL(g_cal[tid].XMaxSpeed);
      ta := INT_TO_REAL(g_cal[tid].XAccelTime) / 10.0;
      td := INT_TO_REAL(g_cal[tid].XDecelTime) / 10.0;
      d_acc := 0.5 * vm * ta;
      d_dec := 0.5 * vm * td;

      (* --- Lift and sink times per station --- *)
      FOR si := MIN_StationIndex TO last_stn DO
        idx_i := si - MIN_StationIndex + 1;
        IF idx_i >= 1 AND idx_i <= 30 THEN
          IF g_station[si].DryWet = 1 THEN
            (* Wet station *)
            g_move[tid].LiftTime[idx_i] := g_cal[tid].LiftWetTime;
            g_move[tid].SinkTime[idx_i] := g_cal[tid].SinkWetTime;
          ELSE
            (* Dry station *)
            g_move[tid].LiftTime[idx_i] := g_cal[tid].LiftDryTime;
            g_move[tid].SinkTime[idx_i] := g_cal[tid].SinkDryTime;
          END_IF;
        END_IF;
      END_FOR;

      (* --- Travel times between stations --- *)
      FOR si := MIN_StationIndex TO last_stn DO
        idx_i := si - MIN_StationIndex + 1;
        IF idx_i >= 1 AND idx_i <= 30 THEN
          FOR sj := MIN_StationIndex TO last_stn DO
            idx_j := sj - MIN_StationIndex + 1;
            IF idx_j >= 1 AND idx_j <= 30 THEN
              IF si = sj THEN
                g_move[tid].Travel[idx_i].ToTime[idx_j] := 0;
              ELSE
                dist := ABS(DINT_TO_REAL(g_station[si].XPosition - g_station[sj].XPosition));
                IF dist < 1.0 THEN
                  t_time := 0.0;
                ELSIF dist >= d_acc + d_dec THEN
                  (* Trapezoidal profile: full accel + cruise + full decel *)
                  t_time := ta + (dist - d_acc - d_dec) / vm + td;
                ELSE
                  (* Triangle profile: cannot reach full speed *)
                  IF ta + td > 0.0 THEN
                    v_peak := SQRT(2.0 * dist * vm / (ta + td));
                    t_time := v_peak * (ta + td) / vm;
                  ELSE
                    t_time := 0.0;
                  END_IF;
                END_IF;
                g_move[tid].Travel[idx_i].ToTime[idx_j] := REAL_TO_INT(t_time * 10.0);
              END_IF;
            END_IF;
          END_FOR;
        END_IF;
      END_FOR;

    END_IF;  (* valid calibration check *)
  END_FOR;

END_IF;

prev_run := i_run;

END_FUNCTION_BLOCK
